LIN {X 0,Y 250.242,Z 442.898,A -85,B 0,C 180,E1 -18826.312,E2 -18826.312} C_VEL
LIN {X 0,Y 252.616,Z 436.287,A -85,B 0,C 180,E1 -18829.075,E2 -18829.075} C_VEL
LIN {X 0,Y 255.174,Z 429.183,A -85,B 0,C 180,E1 -18831.404,E2 -18831.404} C_VEL
LIN {X 0,Y 258.417,Z 420.356,A -85,B 0,C 180,E1 -18833.651,E2 -18833.651} C_VEL
LIN {X 0,Y 261.758,Z 410.378,A -85,B 0,C 180,E1 -18835.655,E2 -18835.655} C_VEL
LIN {X 0,Y 265.23,Z 399.079,A -85,B 0,C 180,E1 -18837.414,E2 -18837.414} C_VEL
LIN {X 0,Y 268.306,Z 387.871,A -85,B 0,C 180,E1 -18838.772,E2 -18838.772} C_VEL
LIN {X 0,Y 271.247,Z 375.163,A -85,B 0,C 180,E1 -18839.919,E2 -18839.919} C_VEL
LIN {X 0,Y 273.533,Z 362.414,A -85,B 0,C 180,E1 -18840.762,E2 -18840.762} C_VEL
LIN {X 0,Y 275.094,Z 349.012,A -85,B 0,C 180,E1 -18841.381,E2 -18841.381} C_VEL
LIN {X 0,Y 278.743,Z 306.37,A -85,B 0,C 180,E1 -18842.929,E2 -18842.929} C_VEL
LIN {X 0,Y 278.232,Z 292.635,A -85,B 0,C 180,E1 -18843.854,E2 -18843.854} C_VEL
LIN {X 0,Y 276.686,Z 276.192,A -85,B 0,C 180,E1 -18845.252,E2 -18845.252} C_VEL
LIN {X 0,Y 276.231,Z 273.561,A -85,B 0,C 180,E1 -18845.549,E2 -18845.549} C_VEL
LIN {X 0,Y 272.855,Z 266.156,A -85,B 0,C 180,E1 -18847.014,E2 -18847.014} C_VEL
LIN {X 0,Y 270.376,Z 261.218,A -85,B 0,C 180,E1 -18848.169,E2 -18848.169} C_VEL
LIN {X 0,Y 267.241,Z 255.568,A -85,B 0,C 180,E1 -18849.719,E2 -18849.719} C_VEL
LIN {X 0,Y 264.068,Z 250.117,A -85,B 0,C 180,E1 -18851.565,E2 -18851.565} C_VEL
LIN {X 0,Y 262.47,Z 244.735,A -85,B 0,C 180,E1 -18854.899,E2 -18854.899} C_VEL
LIN {X 0,Y 261.284,Z 241.259,A -85,B 0,C 180,E1 -18857.743,E2 -18857.743} C_VEL
LIN {X 0,Y 260.601,Z 239.385,A -85,B 0,C 180,E1 -18859.665,E2 -18859.665} C_VEL
LIN {X 0,Y 259.611,Z 236.801,A -85,B 0,C 180,E1 -18863.446,E2 -18863.446} C_VEL
LIN {X 0,Y 259.313,Z 236.04,A -85,B 0,C 180,E1 -18865.308,E2 -18865.308} C_VEL
LIN {X 0,Y 259.034,Z 235.596,A -85,B 0,C 180,E1 -18868.968,E2 -18868.968} C_VEL
LIN {X 0,Y 259.56,Z 236.51,A -85,B 0,C 180,E1 -18873.321,E2 -18873.321} C_VEL
LIN {X 0,Y 260.212,Z 238.641,A -85,B 0,C 180,E1 -18876.679,E2 -18876.679} C_VEL
LIN {X 0,Y 261.471,Z 242.04,A -85,B 0,C 180,E1 -18880.18,E2 -18880.18} C_VEL
LIN {X 0,Y 265.902,Z 248.153,A -85,B 0,C 180,E1 -18882.889,E2 -18882.889} C_VEL
LIN {X 0,Y 269.447,Z 253.421,A -85,B 0,C 180,E1 -18884.716,E2 -18884.716} C_VEL
LIN {X 0,Y 272.549,Z 258.468,A -85,B 0,C 180,E1 -18886.185,E2 -18886.185} C_VEL
LIN {X 0,Y 276.457,Z 265.391,A -85,B 0,C 180,E1 -18887.857,E2 -18887.857} C_VEL
LIN {X 0,Y 280.029,Z 273.175,A -85,B 0,C 180,E1 -18889.352,E2 -18889.352} C_VEL
LIN {X 0,Y 280.54,Z 277.359,A -85,B 0,C 180,E1 -18889.756,E2 -18889.756} C_VEL
LIN {X 0,Y 275.476,Z 327.139,A -85,B 0,C 180,E1 -18891.841,E2 -18891.841} C_VEL
LIN {X 0,Y 273.989,Z 339.798,A -85,B 0,C 180,E1 -18892.631,E2 -18892.631} C_VEL
LIN {X 0,Y 271.988,Z 352.049,A -85,B 0,C 180,E1 -18893.695,E2 -18893.695} C_VEL
LIN {X 0,Y 269.693,Z 362.869,A -85,B 0,C 180,E1 -18894.936,E2 -18894.936} C_VEL
LIN {X 0,Y 266.918,Z 373.483,A -85,B 0,C 180,E1 -18896.519,E2 -18896.519} C_VEL
LIN {X 0,Y 264.386,Z 381.823,A -85,B 0,C 180,E1 -18898.095,E2 -18898.095} C_VEL
LIN {X 0,Y 261.552,Z 389.85,A -85,B 0,C 180,E1 -18899.999,E2 -18899.999} C_VEL
LIN {X 0,Y 259.077,Z 396.31,A -85,B 0,C 180,E1 -18901.942,E2 -18901.942} C_VEL
LIN {X 0,Y 256.732,Z 401.481,A -85,B 0,C 180,E1 -18903.923,E2 -18903.923} C_VEL
LIN {X 0,Y 254.323,Z 406.197,A -85,B 0,C 180,E1 -18906.345,E2 -18906.345} C_VEL
LIN {X 0,Y 252.936,Z 408.542,A -85,B 0,C 180,E1 -18907.985,E2 -18907.985} C_VEL
LIN {X 0,Y 251.736,Z 410.331,A -85,B 0,C 180,E1 -18909.642,E2 -18909.642} C_VEL
LIN {X 0,Y 250.71,Z 411.505,A -85,B 0,C 180,E1 -18911.316,E2 -18911.316} C_VEL
LIN {X 0,Y 249.799,Z 412.162,A -85,B 0,C 180,E1 -18913.007,E2 -18913.007} C_VEL
LIN {X 0,Y 249.072,Z 412.229,A -85,B 0,C 180,E1 -18914.711,E2 -18914.711} C_VEL
LIN {X 0,Y 248.491,Z 411.75,A -85,B 0,C 180,E1 -18916.428,E2 -18916.428} C_VEL
LIN {X 0,Y 248.081,Z 410.706,A -85,B 0,C 180,E1 -18918.156,E2 -18918.156} C_VEL
LIN {X 0,Y 247.752,Z 408.241,A -85,B 0,C 180,E1 -18920.59,E2 -18920.59} C_VEL
LIN {X 0,Y 247.79,Z 403.869,A -85,B 0,C 180,E1 -18923.395,E2 -18923.395} C_VEL
LIN {X 0,Y 248.137,Z 398.052,A -85,B 0,C 180,E1 -18926.04,E2 -18926.04} C_VEL
LIN {X 0,Y 248.571,Z 391.701,A -85,B 0,C 180,E1 -18928.266,E2 -18928.266} C_VEL
LIN {X 0,Y 249.183,Z 383.577,A -85,B 0,C 180,E1 -18930.508,E2 -18930.508} C_VEL
LIN {X 0,Y 249.995,Z 374.485,A -85,B 0,C 180,E1 -18932.5,E2 -18932.5} C_VEL
LIN {X 0,Y 250.841,Z 364.034,A -85,B 0,C 180,E1 -18934.322,E2 -18934.322} C_VEL
LIN {X 0,Y 251.742,Z 352.485,A -85,B 0,C 180,E1 -18935.892,E2 -18935.892} C_VEL
LIN {X 0,Y 252.544,Z 339.639,A -85,B 0,C 180,E1 -18937.198,E2 -18937.198} C_VEL
LIN {X 0,Y 253.177,Z 325.928,A -85,B 0,C 180,E1 -18938.175,E2 -18938.175} C_VEL
LIN {X 0,Y 253.707,Z 305.907,A -85,B 0,C 180,E1 -18939.049,E2 -18939.049} C_VEL
LIN {X 0,Y 255.237,Z 260.217,A -85,B 0,C 180,E1 -18940.855,E2 -18940.855} C_VEL
LIN {X 0,Y 252.11,Z 234.672,A -85,B 0,C 180,E1 -18942.111,E2 -18942.111} C_VEL
LIN {X 0,Y 252.252,Z 229.715,A -85,B 0,C 180,E1 -18943.581,E2 -18943.581} C_VEL
LIN {X 0,Y 250.22,Z 219.034,A -85,B 0,C 180,E1 -18947.121,E2 -18947.121} C_VEL
LIN {X 0,Y 249.092,Z 213.695,A -85,B 0,C 180,E1 -18949.004,E2 -18949.004} C_VEL
LIN {X 0,Y 249.072,Z 213.461,A -85,B 0,C 180,E1 -18949.626,E2 -18949.626} C_VEL
LIN {X 0,Y 249.057,Z 213.463,A -85,B 0,C 180,E1 -18953.658,E2 -18953.658} C_VEL
LIN {X 0,Y 249.038,Z 213.464,A -85,B 0,C 180,E1 -18957.844,E2 -18957.844} C_VEL
LIN {X 0,Y 249.096,Z 213.458,A -85,B 0,C 180,E1 -18961.337,E2 -18961.337} C_VEL
LIN {X 0,Y 249.151,Z 213.448,A -85,B 0,C 180,E1 -18964.967,E2 -18964.967} C_VEL
LIN {X 0,Y 249.109,Z 213.453,A -85,B 0,C 180,E1 -18970.21,E2 -18970.21} C_VEL
LIN {X 0,Y 249.241,Z 213.437,A -85,B 0,C 180,E1 -18973.621,E2 -18973.621} C_VEL
LIN {X 0,Y 249.251,Z 213.435,A -85,B 0,C 180,E1 -18978.615,E2 -18978.615} C_VEL
LIN {X 0,Y 249.482,Z 213.405,A -85,B 0,C 180,E1 -18981.902,E2 -18981.902} C_VEL
LIN {X 0,Y 249.435,Z 213.414,A -85,B 0,C 180,E1 -18986.768,E2 -18986.768} C_VEL
LIN {X 0,Y 249.726,Z 213.374,A -85,B 0,C 180,E1 -18989.999,E2 -18989.999} C_VEL
LIN {X 0,Y 249.434,Z 213.415,A -85,B 0,C 180,E1 -18993.229,E2 -18993.229} C_VEL
LIN {X 0,Y 249.476,Z 213.404,A -85,B 0,C 180,E1 -18998.096,E2 -18998.096} C_VEL
LIN {X 0,Y 249.249,Z 213.436,A -85,B 0,C 180,E1 -19001.382,E2 -19001.382} C_VEL
LIN {X 0,Y 249.238,Z 213.436,A -85,B 0,C 180,E1 -19006.377,E2 -19006.377} C_VEL
LIN {X 0,Y 249.082,Z 213.456,A -85,B 0,C 180,E1 -19011.517,E2 -19011.517} C_VEL
LIN {X 0,Y 249.126,Z 213.449,A -85,B 0,C 180,E1 -19015.482,E2 -19015.482} C_VEL
LIN {X 0,Y 249.078,Z 213.458,A -85,B 0,C 180,E1 -19018.993,E2 -19018.993} C_VEL
LIN {X 0,Y 249.03,Z 213.465,A -85,B 0,C 180,E1 -19022.424,E2 -19022.424} C_VEL
LIN {X 0,Y 249.069,Z 213.46,A -85,B 0,C 180,E1 -19026.337,E2 -19026.337} C_VEL
LIN {X 0,Y 249.071,Z 213.459,A -85,B 0,C 180,E1 -19030.463,E2 -19030.463} C_VEL
LIN {X 0,Y 249.015,Z 213.465,A -85,B 0,C 180,E1 -19034.874,E2 -19034.874} C_VEL
LIN {X 0,Y 249.047,Z 213.46,A -85,B 0,C 180,E1 -19037.37,E2 -19037.37} C_VEL
LIN {X 0,Y 249.058,Z 213.462,A -85,B 0,C 180,E1 -19042.193,E2 -19042.193} C_VEL
LIN {X 0,Y 249.055,Z 213.46,A -85,B 0,C 180,E1 -19045.642,E2 -19045.642} C_VEL
LIN {X 0,Y 249.044,Z 213.459,A -85,B 0,C 180,E1 -19049.473,E2 -19049.473} C_VEL
LIN {X 0,Y 249.066,Z 213.458,A -85,B 0,C 180,E1 -19053.162,E2 -19053.162} C_VEL
LIN {X 0,Y 249.072,Z 213.455,A -85,B 0,C 180,E1 -19056.733,E2 -19056.733} C_VEL
LIN {X 0,Y 249.104,Z 213.456,A -85,B 0,C 180,E1 -19060.212,E2 -19060.212} C_VEL
LIN {X 0,Y 249.235,Z 213.439,A -85,B 0,C 180,E1 -19063.622,E2 -19063.622} C_VEL
LIN {X 0,Y 249.237,Z 213.437,A -85,B 0,C 180,E1 -19068.617,E2 -19068.617} C_VEL
LIN {X 0,Y 249.448,Z 213.413,A -85,B 0,C 180,E1 -19071.903,E2 -19071.903} C_VEL
LIN {X 0,Y 249.289,Z 213.429,A -85,B 0,C 180,E1 -19075.149,E2 -19075.149} C_VEL
LIN {X 0,Y 249.669,Z 213.383,A -85,B 0,C 180,E1 -19078.388,E2 -19078.388} C_VEL
LIN {X 0,Y 249.669,Z 213.385,A -85,B 0,C 180,E1 -19081.614,E2 -19081.614} C_VEL
LIN {X 0,Y 249.454,Z 213.41,A -85,B 0,C 180,E1 -19086.471,E2 -19086.471} C_VEL
LIN {X 0,Y 249.383,Z 213.419,A -85,B 0,C 180,E1 -19089.736,E2 -19089.736} C_VEL
LIN {X 0,Y 249.2,Z 213.442,A -85,B 0,C 180,E1 -19094.704,E2 -19094.704} C_VEL
LIN {X 0,Y 249.134,Z 213.448,A -85,B 0,C 180,E1 -19098.078,E2 -19098.078} C_VEL
LIN {X 0,Y 249.082,Z 213.459,A -85,B 0,C 180,E1 -19101.519,E2 -19101.519} C_VEL
LIN {X 0,Y 249.073,Z 213.457,A -85,B 0,C 180,E1 -19103.868,E2 -19103.868} C_VEL
LIN {X 0,Y 248.416,Z 213.543,A -85,B 0,C 180,E1 -19105.217,E2 -19105.217} C_VEL
LIN {X 0,Y 245.523,Z 213.901,A -85,B 0,C 180,E1 -19107.414,E2 -19107.414} C_VEL
LIN {X 0,Y 243.064,Z 214.209,A -85,B 0,C 180,E1 -19109.205,E2 -19109.205} C_VEL
LIN {X 0,Y 242.026,Z 214.336,A -85,B 0,C 180,E1 -19110.595,E2 -19110.595} C_VEL
LIN {X 0,Y 241.952,Z 214.342,A -85,B 0,C 180,E1 -19111.066,E2 -19111.066} C_VEL
LIN {X 0,Y 242.002,Z 214.339,A -85,B 0,C 180,E1 -19115.598,E2 -19115.598} C_VEL
LIN {X 0,Y 241.953,Z 214.345,A -85,B 0,C 180,E1 -19119.721,E2 -19119.721} C_VEL
LIN {X 0,Y 241.916,Z 214.349,A -85,B 0,C 180,E1 -19124.206,E2 -19124.206} C_VEL
LIN {X 0,Y 241.932,Z 214.348,A -85,B 0,C 180,E1 -19128.079,E2 -19128.079} C_VEL
LIN {X 0,Y 242.039,Z 214.525,A -85,B 0,C 180,E1 -19132.235,E2 -19132.235} C_VEL
LIN {X 0,Y 245.004,Z 227.718,A -85,B 0,C 180,E1 -19136.293,E2 -19136.293} C_VEL
LIN {X 0,Y 247.94,Z 241.383,A -85,B 0,C 180,E1 -19140.263,E2 -19140.263} C_VEL
LIN {X 0,Y 248.195,Z 243.179,A -85,B 0,C 180,E1 -19140.762,E2 -19140.762} C_VEL
LIN {X 0,Y 246.035,Z 256.439,A -85,B 0,C 180,E1 -19144.177,E2 -19144.177} C_VEL
LIN {X 0,Y 247.085,Z 277.97,A -85,B 0,C 180,E1 -19145.106,E2 -19145.106} C_VEL
LIN {X 0,Y 248.735,Z 300.915,A -85,B 0,C 180,E1 -19146.066,E2 -19146.066} C_VEL
LIN {X 0,Y 247.023,Z 359.054,A -85,B 0,C 180,E1 -19148.24,E2 -19148.24} C_VEL
LIN {X 0,Y 246.323,Z 371.481,A -85,B 0,C 180,E1 -19148.998,E2 -19148.998} C_VEL
LIN {X 0,Y 245.403,Z 383.203,A -85,B 0,C 180,E1 -19150.01,E2 -19150.01} C_VEL
LIN {X 0,Y 244.335,Z 394.661,A -85,B 0,C 180,E1 -19151.339,E2 -19151.339} C_VEL
LIN {X 0,Y 243.271,Z 405.628,A -85,B 0,C 180,E1 -19152.962,E2 -19152.962} C_VEL
LIN {X 0,Y 242.195,Z 415.752,A -85,B 0,C 180,E1 -19154.862,E2 -19154.862} C_VEL
LIN {X 0,Y 241.442,Z 424.766,A -85,B 0,C 180,E1 -19156.964,E2 -19156.964} C_VEL
LIN {X 0,Y 240.968,Z 432.123,A -85,B 0,C 180,E1 -19159.073,E2 -19159.073} C_VEL
LIN {X 0,Y 240.761,Z 439.176,A -85,B 0,C 180,E1 -19161.609,E2 -19161.609} C_VEL
LIN {X 0,Y 240.805,Z 444.675,A -85,B 0,C 180,E1 -19164.138,E2 -19164.138} C_VEL
LIN {X 0,Y 240.983,Z 448.811,A -85,B 0,C 180,E1 -19166.657,E2 -19166.657} C_VEL
LIN {X 0,Y 241.109,Z 450.863,A -85,B 0,C 180,E1 -19168.331,E2 -19168.331} C_VEL
LIN {X 0,Y 241.116,Z 452.378,A -85,B 0,C 180,E1 -19170.001,E2 -19170.001} C_VEL
LIN {X 0,Y 240.997,Z 453.423,A -85,B 0,C 180,E1 -19171.672,E2 -19171.672} C_VEL
LIN {X 0,Y 240.622,Z 453.947,A -85,B 0,C 180,E1 -19173.35,E2 -19173.35} C_VEL
LIN {X 0,Y 240.281,Z 453.905,A -85,B 0,C 180,E1 -19176.022,E2 -19176.022} C_VEL
LIN {X 0,Y 240.213,Z 452.989,A -85,B 0,C 180,E1 -19178.413,E2 -19178.413} C_VEL
LIN {X 0,Y 240.738,Z 450.239,A -85,B 0,C 180,E1 -19181.793,E2 -19181.793} C_VEL
LIN {X 0,Y 241.879,Z 447.064,A -85,B 0,C 180,E1 -19184.3,E2 -19184.3} C_VEL
LIN {X 0,Y 243.423,Z 442.874,A -85,B 0,C 180,E1 -19186.782,E2 -19186.782} C_VEL
LIN {X 0,Y 245.831,Z 436.744,A -85,B 0,C 180,E1 -19189.547,E2 -19189.547} C_VEL
LIN {X 0,Y 248.587,Z 429.654,A -85,B 0,C 180,E1 -19192.001,E2 -19192.001} C_VEL
LIN {X 0,Y 251.986,Z 421.175,A -85,B 0,C 180,E1 -19194.293,E2 -19194.293} C_VEL
LIN {X 0,Y 255.123,Z 412.586,A -85,B 0,C 180,E1 -19196.153,E2 -19196.153} C_VEL
LIN {X 0,Y 258.683,Z 402.079,A -85,B 0,C 180,E1 -19197.948,E2 -19197.948} C_VEL
LIN {X 0,Y 261.804,Z 391.752,A -85,B 0,C 180,E1 -19199.336,E2 -19199.336} C_VEL
LIN {X 0,Y 265.258,Z 378.523,A -85,B 0,C 180,E1 -19200.667,E2 -19200.667} C_VEL
LIN {X 0,Y 267.695,Z 366.659,A -85,B 0,C 180,E1 -19201.564,E2 -19201.564} C_VEL
LIN {X 0,Y 269.831,Z 352.408,A -85,B 0,C 180,E1 -19202.328,E2 -19202.328} C_VEL
LIN {X 0,Y 273.994,Z 306.663,A -85,B 0,C 180,E1 -19204.05,E2 -19204.05} C_VEL
LIN {X 0,Y 273.515,Z 292.928,A -85,B 0,C 180,E1 -19205.03,E2 -19205.03} C_VEL
LIN {X 0,Y 272.25,Z 277.749,A -85,B 0,C 180,E1 -19206.404,E2 -19206.404} C_VEL
LIN {X 0,Y 269.163,Z 270.902,A -85,B 0,C 180,E1 -19207.837,E2 -19207.837} C_VEL
LIN {X 0,Y 266.967,Z 266.304,A -85,B 0,C 180,E1 -19208.942,E2 -19208.942} C_VEL
LIN {X 0,Y 264.32,Z 261.353,A -85,B 0,C 180,E1 -19210.347,E2 -19210.347} C_VEL
LIN {X 0,Y 260.674,Z 255.2,A -85,B 0,C 180,E1 -19212.513,E2 -19212.513} C_VEL
LIN {X 0,Y 256.954,Z 248.907,A -85,B 0,C 180,E1 -19215.328,E2 -19215.328} C_VEL
LIN {X 0,Y 255.623,Z 245.043,A -85,B 0,C 180,E1 -19218.711,E2 -19218.711} C_VEL
LIN {X 0,Y 254.553,Z 242.132,A -85,B 0,C 180,E1 -19222.597,E2 -19222.597} C_VEL
LIN {X 0,Y 254.253,Z 241.129,A -85,B 0,C 180,E1 -19224.515,E2 -19224.515} C_VEL
LIN {X 0,Y 253.852,Z 240.45,A -85,B 0,C 180,E1 -19229.122,E2 -19229.122} C_VEL
LIN {X 0,Y 254.111,Z 240.979,A -85,B 0,C 180,E1 -19232.256,E2 -19232.256} C_VEL
LIN {X 0,Y 254.384,Z 241.552,A -85,B 0,C 180,E1 -19233.765,E2 -19233.765} C_VEL
LIN {X 0,Y 255.017,Z 243.339,A -85,B 0,C 180,E1 -19236.387,E2 -19236.387} C_VEL
LIN {X 0,Y 259.406,Z 248.969,A -85,B 0,C 180,E1 -19239.974,E2 -19239.974} C_VEL
LIN {X 0,Y 263.342,Z 254.427,A -85,B 0,C 180,E1 -19242.435,E2 -19242.435} C_VEL
LIN {X 0,Y 266.413,Z 259.247,A -85,B 0,C 180,E1 -19244.128,E2 -19244.128} C_VEL
LIN {X 0,Y 269.216,Z 263.882,A -85,B 0,C 180,E1 -19245.514,E2 -19245.514} C_VEL
LIN {X 0,Y 273.059,Z 271.072,A -85,B 0,C 180,E1 -19247.297,E2 -19247.297} C_VEL
LIN {X 0,Y 275.758,Z 277.511,A -85,B 0,C 180,E1 -19248.545,E2 -19248.545} C_VEL
LIN {X 0,Y 275.789,Z 279.841,A -85,B 0,C 180,E1 -19248.723,E2 -19248.723} C_VEL
LIN {X 0,Y 270.622,Z 328.589,A -85,B 0,C 180,E1 -19250.802,E2 -19250.802} C_VEL
LIN {X 0,Y 268.929,Z 341.564,A -85,B 0,C 180,E1 -19251.641,E2 -19251.641} C_VEL
LIN {X 0,Y 266.965,Z 352.562,A -85,B 0,C 180,E1 -19252.626,E2 -19252.626} C_VEL
LIN {X 0,Y 264.468,Z 363.457,A -85,B 0,C 180,E1 -19253.897,E2 -19253.897} C_VEL
LIN {X 0,Y 261.219,Z 375.14,A -85,B 0,C 180,E1 -19255.676,E2 -19255.676} C_VEL
LIN {X 0,Y 258.565,Z 383.268,A -85,B 0,C 180,E1 -19257.273,E2 -19257.273} C_VEL
LIN {X 0,Y 255.535,Z 391.182,A -85,B 0,C 180,E1 -19259.211,E2 -19259.211} C_VEL
LIN {X 0,Y 253.054,Z 397.105,A -85,B 0,C 180,E1 -19261.065,E2 -19261.065} C_VEL
LIN {X 0,Y 250.411,Z 402.538,A -85,B 0,C 180,E1 -19263.217,E2 -19263.217} C_VEL
LIN {X 0,Y 248.03,Z 406.89,A -85,B 0,C 180,E1 -19265.509,E2 -19265.509} C_VEL
LIN {X 0,Y 245.68,Z 410.416,A -85,B 0,C 180,E1 -19268.222,E2 -19268.222} C_VEL
LIN {X 0,Y 244.462,Z 411.843,A -85,B 0,C 180,E1 -19269.932,E2 -19269.932} C_VEL
LIN {X 0,Y 243.43,Z 412.692,A -85,B 0,C 180,E1 -19271.659,E2 -19271.659} C_VEL
LIN {X 0,Y 242.549,Z 413.034,A -85,B 0,C 180,E1 -19273.402,E2 -19273.402} C_VEL
LIN {X 0,Y 241.491,Z 412.383,A -85,B 0,C 180,E1 -19276.18,E2 -19276.18} C_VEL
LIN {X 0,Y 240.877,Z 410.594,A -85,B 0,C 180,E1 -19278.719,E2 -19278.719} C_VEL
LIN {X 0,Y 240.632,Z 407.265,A -85,B 0,C 180,E1 -19281.493,E2 -19281.493} C_VEL
LIN {X 0,Y 240.773,Z 402.698,A -85,B 0,C 180,E1 -19284.119,E2 -19284.119} C_VEL
LIN {X 0,Y 241.108,Z 397.438,A -85,B 0,C 180,E1 -19286.392,E2 -19286.392} C_VEL
LIN {X 0,Y 241.669,Z 389.71,A -85,B 0,C 180,E1 -19288.984,E2 -19288.984} C_VEL
LIN {X 0,Y 242.241,Z 382.109,A -85,B 0,C 180,E1 -19290.995,E2 -19290.995} C_VEL
LIN {X 0,Y 243.1,Z 372.57,A -85,B 0,C 180,E1 -19293.029,E2 -19293.029} C_VEL
LIN {X 0,Y 244.04,Z 361.305,A -85,B 0,C 180,E1 -19294.915,E2 -19294.915} C_VEL
LIN {X 0,Y 244.911,Z 349.633,A -85,B 0,C 180,E1 -19296.422,E2 -19296.422} C_VEL
LIN {X 0,Y 245.629,Z 337.82,A -85,B 0,C 180,E1 -19297.574,E2 -19297.574} C_VEL
LIN {X 0,Y 246.218,Z 324.894,A -85,B 0,C 180,E1 -19298.473,E2 -19298.473} C_VEL
LIN {X 0,Y 246.945,Z 299.704,A -85,B 0,C 180,E1 -19299.574,E2 -19299.574} C_VEL
LIN {X 0,Y 248.312,Z 260.898,A -85,B 0,C 180,E1 -19301.163,E2 -19301.163} C_VEL
LIN {X 0,Y 245.18,Z 235.277,A -85,B 0,C 180,E1 -19302.436,E2 -19302.436} C_VEL
LIN {X 0,Y 245.269,Z 233.089,A -85,B 0,C 180,E1 -19302.999,E2 -19302.999} C_VEL
LIN {X 0,Y 245.025,Z 229.434,A -85,B 0,C 180,E1 -19304.186,E2 -19304.186} C_VEL
LIN {X 0,Y 242.968,Z 219.033,A -85,B 0,C 180,E1 -19307.737,E2 -19307.737} C_VEL
LIN {X 0,Y 242.072,Z 214.513,A -85,B 0,C 180,E1 -19309.394,E2 -19309.394} C_VEL
LIN {X 0,Y 241.99,Z 214.341,A -85,B 0,C 180,E1 -19312.417,E2 -19312.417} C_VEL
LIN {X 0,Y 241.987,Z 214.341,A -85,B 0,C 180,E1 -19316.507,E2 -19316.507} C_VEL
LIN {X 0,Y 242.036,Z 214.334,A -85,B 0,C 180,E1 -19320.586,E2 -19320.586} C_VEL
LIN {X 0,Y 242.067,Z 214.33,A -85,B 0,C 180,E1 -19324.182,E2 -19324.182} C_VEL
LIN {X 0,Y 242.052,Z 214.331,A -85,B 0,C 180,E1 -19328.296,E2 -19328.296} C_VEL
LIN {X 0,Y 242.162,Z 214.32,A -85,B 0,C 180,E1 -19333.277,E2 -19333.277} C_VEL
LIN {X 0,Y 242.185,Z 214.315,A -85,B 0,C 180,E1 -19338.279,E2 -19338.279} C_VEL
LIN {X 0,Y 242.433,Z 214.284,A -85,B 0,C 180,E1 -19341.665,E2 -19341.665} C_VEL
LIN {X 0,Y 242.26,Z 214.309,A -85,B 0,C 180,E1 -19345.006,E2 -19345.006} C_VEL
LIN {X 0,Y 242.634,Z 214.258,A -85,B 0,C 180,E1 -19348.339,E2 -19348.339} C_VEL
LIN {X 0,Y 242.634,Z 214.259,A -85,B 0,C 180,E1 -19351.659,E2 -19351.659} C_VEL
LIN {X 0,Y 242.428,Z 214.286,A -85,B 0,C 180,E1 -19356.658,E2 -19356.658} C_VEL
LIN {X 0,Y 242.311,Z 214.299,A -85,B 0,C 180,E1 -19360.021,E2 -19360.021} C_VEL
LIN {X 0,Y 242.163,Z 214.318,A -85,B 0,C 180,E1 -19365.14,E2 -19365.14} C_VEL
LIN {X 0,Y 242.069,Z 214.331,A -85,B 0,C 180,E1 -19368.623,E2 -19368.623} C_VEL
LIN {X 0,Y 242.008,Z 214.338,A -85,B 0,C 180,E1 -19372.179,E2 -19372.179} C_VEL
LIN {X 0,Y 242.061,Z 214.329,A -85,B 0,C 180,E1 -19375.837,E2 -19375.837} C_VEL
LIN {X 0,Y 242.025,Z 214.335,A -85,B 0,C 180,E1 -19379.579,E2 -19379.579} C_VEL
LIN {X 0,Y 241.985,Z 214.338,A -85,B 0,C 180,E1 -19383.49,E2 -19383.49} C_VEL
LIN {X 0,Y 242.007,Z 214.337,A -85,B 0,C 180,E1 -19387.577,E2 -19387.577} C_VEL
LIN {X 0,Y 241.978,Z 214.339,A -85,B 0,C 180,E1 -19391.912,E2 -19391.912} C_VEL
LIN {X 0,Y 241.98,Z 214.343,A -85,B 0,C 180,E1 -19396.558,E2 -19396.558} C_VEL
LIN {X 0,Y 241.975,Z 214.343,A -85,B 0,C 180,E1 -19400.286,E2 -19400.286} C_VEL
LIN {X 0,Y 242.03,Z 214.337,A -85,B 0,C 180,E1 -19404.497,E2 -19404.497} C_VEL
LIN {X 0,Y 241.969,Z 214.342,A -85,B 0,C 180,E1 -19408.48,E2 -19408.48} C_VEL
LIN {X 0,Y 242,Z 214.341,A -85,B 0,C 180,E1 -19412.313,E2 -19412.313} C_VEL
LIN {X 0,Y 242.05,Z 214.334,A -85,B 0,C 180,E1 -19416.016,E2 -19416.016} C_VEL
LIN {X 0,Y 242.03,Z 214.335,A -85,B 0,C 180,E1 -19419.608,E2 -19419.608} C_VEL
LIN {X 0,Y 242.156,Z 214.319,A -85,B 0,C 180,E1 -19423.279,E2 -19423.279} C_VEL
LIN {X 0,Y 242.174,Z 214.318,A -85,B 0,C 180,E1 -19428.28,E2 -19428.28} C_VEL
LIN {X 0,Y 242.393,Z 214.292,A -85,B 0,C 180,E1 -19431.665,E2 -19431.665} C_VEL
LIN {X 0,Y 242.25,Z 214.306,A -85,B 0,C 180,E1 -19435.008,E2 -19435.008} C_VEL
LIN {X 0,Y 242.629,Z 214.26,A -85,B 0,C 180,E1 -19438.341,E2 -19438.341} C_VEL
LIN {X 0,Y 242.629,Z 214.261,A -85,B 0,C 180,E1 -19441.661,E2 -19441.661} C_VEL
LIN {X 0,Y 242.427,Z 214.285,A -85,B 0,C 180,E1 -19446.66,E2 -19446.66} C_VEL
LIN {X 0,Y 242.308,Z 214.298,A -85,B 0,C 180,E1 -19450.023,E2 -19450.023} C_VEL
LIN {X 0,Y 242.161,Z 214.32,A -85,B 0,C 180,E1 -19455.142,E2 -19455.142} C_VEL
LIN {X 0,Y 242.068,Z 214.328,A -85,B 0,C 180,E1 -19458.625,E2 -19458.625} C_VEL
LIN {X 0,Y 242.008,Z 214.337,A -85,B 0,C 180,E1 -19462.181,E2 -19462.181} C_VEL
LIN {X 0,Y 242.062,Z 214.33,A -85,B 0,C 180,E1 -19465.839,E2 -19465.839} C_VEL
LIN {X 0,Y 242.003,Z 214.34,A -85,B 0,C 180,E1 -19469.585,E2 -19469.585} C_VEL
LIN {X 0,Y 241.952,Z 214.342,A -85,B 0,C 180,E1 -19471.066,E2 -19471.066} C_VEL
LIN {X 0,Y 241.297,Z 214.428,A -85,B 0,C 180,E1 -19472.456,E2 -19472.456} C_VEL
LIN {X 0,Y 238.411,Z 214.787,A -85,B 0,C 180,E1 -19474.722,E2 -19474.722} C_VEL
LIN {X 0,Y 235.968,Z 215.09,A -85,B 0,C 180,E1 -19476.569,E2 -19476.569} C_VEL
LIN {X 0,Y 234.953,Z 215.216,A -85,B 0,C 180,E1 -19478.003,E2 -19478.003} C_VEL
LIN {X 0,Y 234.89,Z 215.223,A -85,B 0,C 180,E1 -19478.489,E2 -19478.489} C_VEL
LIN {X 0,Y 234.878,Z 215.227,A -85,B 0,C 180,E1 -19481.581,E2 -19481.581} C_VEL
LIN {X 0,Y 234.882,Z 215.226,A -85,B 0,C 180,E1 -19485.9,E2 -19485.9} C_VEL
LIN {X 0,Y 234.88,Z 215.229,A -85,B 0,C 180,E1 -19488.834,E2 -19488.834} C_VEL
LIN {X 0,Y 234.993,Z 215.432,A -85,B 0,C 180,E1 -19491.819,E2 -19491.819} C_VEL
LIN {X 0,Y 237.844,Z 228.125,A -85,B 0,C 180,E1 -19495.847,E2 -19495.847} C_VEL
LIN {X 0,Y 240.65,Z 241.145,A -85,B 0,C 180,E1 -19499.752,E2 -19499.752} C_VEL
LIN {X 0,Y 241.062,Z 244.801,A -85,B 0,C 180,E1 -19500.796,E2 -19500.796} C_VEL
LIN {X 0,Y 239.126,Z 256.051,A -85,B 0,C 180,E1 -19503.785,E2 -19503.785} C_VEL
LIN {X 0,Y 240.01,Z 276.708,A -85,B 0,C 180,E1 -19504.714,E2 -19504.714} C_VEL
LIN {X 0,Y 241.754,Z 301.362,A -85,B 0,C 180,E1 -19505.791,E2 -19505.791} C_VEL
LIN {X 0,Y 239.987,Z 358.705,A -85,B 0,C 180,E1 -19508.021,E2 -19508.021} C_VEL
LIN {X 0,Y 239.29,Z 371.062,A -85,B 0,C 180,E1 -19508.802,E2 -19508.802} C_VEL
LIN {X 0,Y 238.473,Z 381.707,A -85,B 0,C 180,E1 -19509.741,E2 -19509.741} C_VEL
LIN {X 0,Y 237.324,Z 393.659,A -85,B 0,C 180,E1 -19511.142,E2 -19511.142} C_VEL
LIN {X 0,Y 236.195,Z 405.3,A -85,B 0,C 180,E1 -19512.914,E2 -19512.914} C_VEL
LIN {X 0,Y 235.134,Z 415.219,A -85,B 0,C 180,E1 -19514.84,E2 -19514.84} C_VEL
LIN {X 0,Y 234.387,Z 424.22,A -85,B 0,C 180,E1 -19517.005,E2 -19517.005} C_VEL
LIN {X 0,Y 233.925,Z 431.56,A -85,B 0,C 180,E1 -19519.178,E2 -19519.178} C_VEL
LIN {X 0,Y 233.723,Z 438.587,A -85,B 0,C 180,E1 -19521.79,E2 -19521.79} C_VEL
LIN {X 0,Y 233.769,Z 443.252,A -85,B 0,C 180,E1 -19523.961,E2 -19523.961} C_VEL
LIN {X 0,Y 233.966,Z 447.567,A -85,B 0,C 180,E1 -19526.557,E2 -19526.557} C_VEL
LIN {X 0,Y 234.069,Z 449.75,A -85,B 0,C 180,E1 -19528.281,E2 -19528.281} C_VEL
LIN {X 0,Y 234.083,Z 451.357,A -85,B 0,C 180,E1 -19530.001,E2 -19530.001} C_VEL
LIN {X 0,Y 233.944,Z 452.461,A -85,B 0,C 180,E1 -19531.723,E2 -19531.723} C_VEL
LIN {X 0,Y 233.568,Z 453.099,A -85,B 0,C 180,E1 -19533.451,E2 -19533.451} C_VEL
LIN {X 0,Y 233.224,Z 453.225,A -85,B 0,C 180,E1 -19536.045,E2 -19536.045} C_VEL
LIN {X 0,Y 233.157,Z 452.402,A -85,B 0,C 180,E1 -19538.669,E2 -19538.669} C_VEL
LIN {X 0,Y 233.36,Z 451.359,A -85,B 0,C 180,E1 -19540.412,E2 -19540.412} C_VEL
LIN {X 0,Y 233.742,Z 449.87,A -85,B 0,C 180,E1 -19542.151,E2 -19542.151} C_VEL
LIN {X 0,Y 234.965,Z 446.886,A -85,B 0,C 180,E1 -19544.73,E2 -19544.73} C_VEL
LIN {X 0,Y 236.627,Z 442.873,A -85,B 0,C 180,E1 -19547.279,E2 -19547.279} C_VEL
LIN {X 0,Y 238.829,Z 437.678,A -85,B 0,C 180,E1 -19549.806,E2 -19549.806} C_VEL
LIN {X 0,Y 242.037,Z 430.2,A -85,B 0,C 180,E1 -19552.628,E2 -19552.628} C_VEL
LIN {X 0,Y 245.589,Z 422.035,A -85,B 0,C 180,E1 -19554.968,E2 -19554.968} C_VEL
LIN {X 0,Y 248.87,Z 413.774,A -85,B 0,C 180,E1 -19556.862,E2 -19556.862} C_VEL
LIN {X 0,Y 252.527,Z 403.736,A -85,B 0,C 180,E1 -19558.692,E2 -19558.692} C_VEL
LIN {X 0,Y 256.173,Z 392.632,A -85,B 0,C 180,E1 -19560.273,E2 -19560.273} C_VEL
LIN {X 0,Y 259.339,Z 381.873,A -85,B 0,C 180,E1 -19561.445,E2 -19561.445} C_VEL
LIN {X 0,Y 262.309,Z 368.985,A -85,B 0,C 180,E1 -19562.517,E2 -19562.517} C_VEL
LIN {X 0,Y 264.556,Z 356.138,A -85,B 0,C 180,E1 -19563.281,E2 -19563.281} C_VEL
LIN {X 0,Y 266.971,Z 333.427,A -85,B 0,C 180,E1 -19564.175,E2 -19564.175} C_VEL
LIN {X 0,Y 269.438,Z 307.883,A -85,B 0,C 180,E1 -19565.167,E2 -19565.167} C_VEL
LIN {X 0,Y 269.118,Z 294.607,A -85,B 0,C 180,E1 -19566.158,E2 -19566.158} C_VEL
LIN {X 0,Y 268.15,Z 281.712,A -85,B 0,C 180,E1 -19567.354,E2 -19567.354} C_VEL
LIN {X 0,Y 264.649,Z 273.323,A -85,B 0,C 180,E1 -19569.208,E2 -19569.208} C_VEL
LIN {X 0,Y 261.35,Z 266.949,A -85,B 0,C 180,E1 -19571.058,E2 -19571.058} C_VEL
LIN {X 0,Y 258.273,Z 261.5,A -85,B 0,C 180,E1 -19573.003,E2 -19573.003} C_VEL
LIN {X 0,Y 254.352,Z 254.93,A -85,B 0,C 180,E1 -19576.038,E2 -19576.038} C_VEL
LIN {X 0,Y 251.07,Z 250.024,A -85,B 0,C 180,E1 -19579.549,E2 -19579.549} C_VEL
LIN {X 0,Y 249.498,Z 247.198,A -85,B 0,C 180,E1 -19582.434,E2 -19582.434} C_VEL
LIN {X 0,Y 249.03,Z 245.889,A -85,B 0,C 180,E1 -19584.928,E2 -19584.928} C_VEL
LIN {X 0,Y 248.775,Z 245.426,A -85,B 0,C 180,E1 -19588.718,E2 -19588.718} C_VEL
LIN {X 0,Y 249.865,Z 246.591,A -85,B 0,C 180,E1 -19591.909,E2 -19591.909} C_VEL
LIN {X 0,Y 252.858,Z 249.7,A -85,B 0,C 180,E1 -19595.812,E2 -19595.812} C_VEL
LIN {X 0,Y 257.209,Z 255.47,A -85,B 0,C 180,E1 -19599.574,E2 -19599.574} C_VEL
LIN {X 0,Y 260.693,Z 260.568,A -85,B 0,C 180,E1 -19601.898,E2 -19601.898} C_VEL
LIN {X 0,Y 263.913,Z 265.887,A -85,B 0,C 180,E1 -19603.792,E2 -19603.792} C_VEL
LIN {X 0,Y 266.213,Z 269.891,A -85,B 0,C 180,E1 -19604.986,E2 -19604.986} C_VEL
LIN {X 0,Y 269.463,Z 276.342,A -85,B 0,C 180,E1 -19606.627,E2 -19606.627} C_VEL
LIN {X 0,Y 271.419,Z 280.946,A -85,B 0,C 180,E1 -19607.564,E2 -19607.564} C_VEL
LIN {X 0,Y 265.924,Z 329.453,A -85,B 0,C 180,E1 -19609.682,E2 -19609.682} C_VEL
LIN {X 0,Y 264.207,Z 341.756,A -85,B 0,C 180,E1 -19610.488,E2 -19610.488} C_VEL
LIN {X 0,Y 262.221,Z 352.548,A -85,B 0,C 180,E1 -19611.445,E2 -19611.445} C_VEL
LIN {X 0,Y 259.444,Z 364.16,A -85,B 0,C 180,E1 -19612.802,E2 -19612.802} C_VEL
LIN {X 0,Y 256.534,Z 374.047,A -85,B 0,C 180,E1 -19614.3,E2 -19614.3} C_VEL
LIN {X 0,Y 253.438,Z 383.063,A -85,B 0,C 180,E1 -19616.034,E2 -19616.034} C_VEL
LIN {X 0,Y 250.194,Z 391.101,A -85,B 0,C 180,E1 -19617.987,E2 -19617.987} C_VEL
LIN {X 0,Y 247.326,Z 397.584,A -85,B 0,C 180,E1 -19619.999,E2 -19619.999} C_VEL
LIN {X 0,Y 244.152,Z 403.662,A -85,B 0,C 180,E1 -19622.474,E2 -19622.474} C_VEL
LIN {X 0,Y 241.385,Z 408.2,A -85,B 0,C 180,E1 -19625.01,E2 -19625.01} C_VEL
LIN {X 0,Y 239.776,Z 410.434,A -85,B 0,C 180,E1 -19626.732,E2 -19626.732} C_VEL
LIN {X 0,Y 238.395,Z 412.097,A -85,B 0,C 180,E1 -19628.476,E2 -19628.476} C_VEL
LIN {X 0,Y 236.524,Z 413.573,A -85,B 0,C 180,E1 -19631.315,E2 -19631.315} C_VEL
LIN {X 0,Y 235.279,Z 413.719,A -85,B 0,C 180,E1 -19633.825,E2 -19633.825} C_VEL
LIN {X 0,Y 234.346,Z 412.806,A -85,B 0,C 180,E1 -19636.325,E2 -19636.325} C_VEL
LIN {X 0,Y 233.701,Z 410.287,A -85,B 0,C 180,E1 -19639.316,E2 -19639.316} C_VEL
LIN {X 0,Y 233.53,Z 406.541,A -85,B 0,C 180,E1 -19642.097,E2 -19642.097} C_VEL
LIN {X 0,Y 233.756,Z 401.223,A -85,B 0,C 180,E1 -19644.892,E2 -19644.892} C_VEL
LIN {X 0,Y 234.141,Z 395.375,A -85,B 0,C 180,E1 -19647.241,E2 -19647.241} C_VEL
LIN {X 0,Y 234.747,Z 387.462,A -85,B 0,C 180,E1 -19649.746,E2 -19649.746} C_VEL
LIN {X 0,Y 235.517,Z 378.43,A -85,B 0,C 180,E1 -19651.982,E2 -19651.982} C_VEL
LIN {X 0,Y 236.349,Z 368.722,A -85,B 0,C 180,E1 -19653.9,E2 -19653.9} C_VEL
LIN {X 0,Y 237.244,Z 358.264,A -85,B 0,C 180,E1 -19655.545,E2 -19655.545} C_VEL
LIN {X 0,Y 238.161,Z 345.721,A -85,B 0,C 180,E1 -19657.064,E2 -19657.064} C_VEL
LIN {X 0,Y 238.835,Z 333.321,A -85,B 0,C 180,E1 -19658.165,E2 -19658.165} C_VEL
LIN {X 0,Y 239.297,Z 320.42,A -85,B 0,C 180,E1 -19658.952,E2 -19658.952} C_VEL
LIN {X 0,Y 241.312,Z 261.059,A -85,B 0,C 180,E1 -19661.492,E2 -19661.492} C_VEL
LIN {X 0,Y 238.22,Z 235.353,A -85,B 0,C 180,E1 -19662.826,E2 -19662.826} C_VEL
LIN {X 0,Y 238.254,Z 232.134,A -85,B 0,C 180,E1 -19663.8,E2 -19663.8} C_VEL
LIN {X 0,Y 236.159,Z 220.985,A -85,B 0,C 180,E1 -19667.672,E2 -19667.672} C_VEL
LIN {X 0,Y 235.051,Z 215.426,A -85,B 0,C 180,E1 -19669.715,E2 -19669.715} C_VEL
LIN {X 0,Y 234.938,Z 215.221,A -85,B 0,C 180,E1 -19673.869,E2 -19673.869} C_VEL
LIN {X 0,Y 234.958,Z 215.219,A -85,B 0,C 180,E1 -19677.423,E2 -19677.423} C_VEL
LIN {X 0,Y 234.952,Z 215.22,A -85,B 0,C 180,E1 -19681.405,E2 -19681.405} C_VEL
LIN {X 0,Y 234.987,Z 215.214,A -85,B 0,C 180,E1 -19685.246,E2 -19685.246} C_VEL
LIN {X 0,Y 235.01,Z 215.21,A -85,B 0,C 180,E1 -19688.969,E2 -19688.969} C_VEL
LIN {X 0,Y 235.095,Z 215.2,A -85,B 0,C 180,E1 -19693.058,E2 -19693.058} C_VEL
LIN {X 0,Y 235.145,Z 215.192,A -85,B 0,C 180,E1 -19697.923,E2 -19697.923} C_VEL
LIN {X 0,Y 235.389,Z 215.163,A -85,B 0,C 180,E1 -19701.413,E2 -19701.413} C_VEL
LIN {X 0,Y 235.404,Z 215.162,A -85,B 0,C 180,E1 -19703.14,E2 -19703.14} C_VEL
LIN {X 0,Y 235.594,Z 215.135,A -85,B 0,C 180,E1 -19708.289,E2 -19708.289} C_VEL
LIN {X 0,Y 235.594,Z 215.136,A -85,B 0,C 180,E1 -19711.708,E2 -19711.708} C_VEL
LIN {X 0,Y 235.399,Z 215.163,A -85,B 0,C 180,E1 -19716.857,E2 -19716.857} C_VEL
LIN {X 0,Y 235.234,Z 215.181,A -85,B 0,C 180,E1 -19720.325,E2 -19720.325} C_VEL
LIN {X 0,Y 235.11,Z 215.195,A -85,B 0,C 180,E1 -19725.605,E2 -19725.605} C_VEL
LIN {X 0,Y 235.004,Z 215.211,A -85,B 0,C 180,E1 -19729.204,E2 -19729.204} C_VEL
LIN {X 0,Y 234.956,Z 215.217,A -85,B 0,C 180,E1 -19732.882,E2 -19732.882} C_VEL
LIN {X 0,Y 234.965,Z 215.217,A -85,B 0,C 180,E1 -19736.656,E2 -19736.656} C_VEL
LIN {X 0,Y 234.927,Z 215.223,A -85,B 0,C 180,E1 -19740.567,E2 -19740.567} C_VEL
LIN {X 0,Y 234.955,Z 215.218,A -85,B 0,C 180,E1 -19744.632,E2 -19744.632} C_VEL
LIN {X 0,Y 234.96,Z 215.216,A -85,B 0,C 180,E1 -19748.951,E2 -19748.951} C_VEL
LIN {X 0,Y 234.959,Z 215.214,A -85,B 0,C 180,E1 -19753.467,E2 -19753.467} C_VEL
LIN {X 0,Y 234.954,Z 215.219,A -85,B 0,C 180,E1 -19756.531,E2 -19756.531} C_VEL
LIN {X 0,Y 234.948,Z 215.215,A -85,B 0,C 180,E1 -19761.086,E2 -19761.086} C_VEL
LIN {X 0,Y 234.954,Z 215.216,A -85,B 0,C 180,E1 -19765.367,E2 -19765.367} C_VEL
LIN {X 0,Y 234.961,Z 215.217,A -85,B 0,C 180,E1 -19770.158,E2 -19770.158} C_VEL
LIN {X 0,Y 234.987,Z 215.214,A -85,B 0,C 180,E1 -19773.794,E2 -19773.794} C_VEL
LIN {X 0,Y 235.004,Z 215.209,A -85,B 0,C 180,E1 -19778.97,E2 -19778.97} C_VEL
LIN {X 0,Y 235.089,Z 215.199,A -85,B 0,C 180,E1 -19783.06,E2 -19783.06} C_VEL
LIN {X 0,Y 235.108,Z 215.201,A -85,B 0,C 180,E1 -19787.923,E2 -19787.923} C_VEL
LIN {X 0,Y 235.324,Z 215.171,A -85,B 0,C 180,E1 -19791.413,E2 -19791.413} C_VEL
LIN {X 0,Y 235.367,Z 215.163,A -85,B 0,C 180,E1 -19793.141,E2 -19793.141} C_VEL
LIN {X 0,Y 235.589,Z 215.138,A -85,B 0,C 180,E1 -19798.291,E2 -19798.291} C_VEL
LIN {X 0,Y 235.589,Z 215.138,A -85,B 0,C 180,E1 -19801.71,E2 -19801.71} C_VEL
LIN {X 0,Y 235.398,Z 215.161,A -85,B 0,C 180,E1 -19806.86,E2 -19806.86} C_VEL
LIN {X 0,Y 235.232,Z 215.178,A -85,B 0,C 180,E1 -19810.328,E2 -19810.328} C_VEL
LIN {X 0,Y 235.108,Z 215.199,A -85,B 0,C 180,E1 -19815.608,E2 -19815.608} C_VEL
LIN {X 0,Y 235.004,Z 215.21,A -85,B 0,C 180,E1 -19819.207,E2 -19819.207} C_VEL
LIN {X 0,Y 234.956,Z 215.217,A -85,B 0,C 180,E1 -19822.884,E2 -19822.884} C_VEL
LIN {X 0,Y 234.963,Z 215.214,A -85,B 0,C 180,E1 -19826.659,E2 -19826.659} C_VEL
LIN {X 0,Y 234.9,Z 215.22,A -85,B 0,C 180,E1 -19831.058,E2 -19831.058} C_VEL
LIN {X 0,Y 234.923,Z 215.221,A -85,B 0,C 180,E1 -19834.64,E2 -19834.64} C_VEL
LIN {X 0,Y 234.89,Z 215.223,A -85,B 0,C 180,E1 -19838.489,E2 -19838.489} C_VEL
LIN {X 0,Y 234.266,Z 215.308,A -85,B 0,C 180,E1 -19839.919,E2 -19839.919} C_VEL
LIN {X 0,Y 231.405,Z 215.666,A -85,B 0,C 180,E1 -19842.251,E2 -19842.251} C_VEL
LIN {X 0,Y 228.937,Z 215.968,A -85,B 0,C 180,E1 -19844.152,E2 -19844.152} C_VEL
LIN {X 0,Y 227.868,Z 216.101,A -85,B 0,C 180,E1 -19845.629,E2 -19845.629} C_VEL
LIN {X 0,Y 227.778,Z 216.109,A -85,B 0,C 180,E1 -19846.13,E2 -19846.13} C_VEL
LIN {X 0,Y 227.934,Z 216.262,A -85,B 0,C 180,E1 -19851.363,E2 -19851.363} C_VEL
LIN {X 0,Y 230.666,Z 228.402,A -85,B 0,C 180,E1 -19855.352,E2 -19855.352} C_VEL
LIN {X 0,Y 233.606,Z 242.159,A -85,B 0,C 180,E1 -19859.605,E2 -19859.605} C_VEL
LIN {X 0,Y 233.945,Z 246.014,A -85,B 0,C 180,E1 -19860.731,E2 -19860.731} C_VEL
LIN {X 0,Y 232.155,Z 255.932,A -85,B 0,C 180,E1 -19863.429,E2 -19863.429} C_VEL
LIN {X 0,Y 233.175,Z 278.937,A -85,B 0,C 180,E1 -19864.481,E2 -19864.481} C_VEL
LIN {X 0,Y 234.75,Z 301.958,A -85,B 0,C 180,E1 -19865.516,E2 -19865.516} C_VEL
LIN {X 0,Y 232.956,Z 358.354,A -85,B 0,C 180,E1 -19867.788,E2 -19867.788} C_VEL
LIN {X 0,Y 232.252,Z 370.631,A -85,B 0,C 180,E1 -19868.593,E2 -19868.593} C_VEL
LIN {X 0,Y 231.45,Z 381.257,A -85,B 0,C 180,E1 -19869.563,E2 -19869.563} C_VEL
LIN {X 0,Y 230.271,Z 393.224,A -85,B 0,C 180,E1 -19871.014,E2 -19871.014} C_VEL
LIN {X 0,Y 229.137,Z 404.784,A -85,B 0,C 180,E1 -19872.831,E2 -19872.831} C_VEL
LIN {X 0,Y 228.059,Z 414.681,A -85,B 0,C 180,E1 -19874.816,E2 -19874.816} C_VEL
LIN {X 0,Y 227.318,Z 423.661,A -85,B 0,C 180,E1 -19877.049,E2 -19877.049} C_VEL
LIN {X 0,Y 226.884,Z 430.97,A -85,B 0,C 180,E1 -19879.29,E2 -19879.29} C_VEL
LIN {X 0,Y 226.701,Z 437.962,A -85,B 0,C 180,E1 -19881.983,E2 -19881.983} C_VEL
LIN {X 0,Y 226.81,Z 443.409,A -85,B 0,C 180,E1 -19884.667,E2 -19884.667} C_VEL
LIN {X 0,Y 226.961,Z 447.47,A -85,B 0,C 180,E1 -19887.339,E2 -19887.339} C_VEL
LIN {X 0,Y 227.057,Z 450.282,A -85,B 0,C 180,E1 -19890.001,E2 -19890.001} C_VEL
LIN {X 0,Y 226.892,Z 451.482,A -85,B 0,C 180,E1 -19891.776,E2 -19891.776} C_VEL
LIN {X 0,Y 226.514,Z 452.197,A -85,B 0,C 180,E1 -19893.559,E2 -19893.559} C_VEL
LIN {X 0,Y 226.157,Z 452.488,A -85,B 0,C 180,E1 -19896.046,E2 -19896.046} C_VEL
LIN {X 0,Y 226.094,Z 451.805,A -85,B 0,C 180,E1 -19898.942,E2 -19898.942} C_VEL
LIN {X 0,Y 226.759,Z 449.516,A -85,B 0,C 180,E1 -19902.531,E2 -19902.531} C_VEL
LIN {X 0,Y 228.068,Z 446.695,A -85,B 0,C 180,E1 -19905.186,E2 -19905.186} C_VEL
LIN {X 0,Y 229.854,Z 442.869,A -85,B 0,C 180,E1 -19907.805,E2 -19907.805} C_VEL
LIN {X 0,Y 232.518,Z 437.135,A -85,B 0,C 180,E1 -19910.757,E2 -19910.757} C_VEL
LIN {X 0,Y 235.53,Z 430.711,A -85,B 0,C 180,E1 -19913.29,E2 -19913.29} C_VEL
LIN {X 0,Y 239.23,Z 422.886,A -85,B 0,C 180,E1 -19915.679,E2 -19915.679} C_VEL
LIN {X 0,Y 243.372,Z 413.227,A -85,B 0,C 180,E1 -19917.987,E2 -19917.987} C_VEL
LIN {X 0,Y 247.256,Z 403.357,A -85,B 0,C 180,E1 -19919.83,E2 -19919.83} C_VEL
LIN {X 0,Y 251.078,Z 392.318,A -85,B 0,C 180,E1 -19921.423,E2 -19921.423} C_VEL
LIN {X 0,Y 254.846,Z 379.883,A -85,B 0,C 180,E1 -19922.767,E2 -19922.767} C_VEL
LIN {X 0,Y 258.016,Z 366.704,A -85,B 0,C 180,E1 -19923.828,E2 -19923.828} C_VEL
LIN {X 0,Y 260.38,Z 353.003,A -85,B 0,C 180,E1 -19924.615,E2 -19924.615} C_VEL
LIN {X 0,Y 265.053,Z 308.913,A -85,B 0,C 180,E1 -19926.353,E2 -19926.353} C_VEL
LIN {X 0,Y 264.816,Z 295.766,A -85,B 0,C 180,E1 -19927.38,E2 -19927.38} C_VEL
LIN {X 0,Y 264.214,Z 285.654,A -85,B 0,C 180,E1 -19928.371,E2 -19928.371} C_VEL
LIN {X 0,Y 261.35,Z 278.505,A -85,B 0,C 180,E1 -19930.004,E2 -19930.004} C_VEL
LIN {X 0,Y 258.559,Z 272.73,A -85,B 0,C 180,E1 -19931.72,E2 -19931.72} C_VEL
LIN {X 0,Y 255.697,Z 267.471,A -85,B 0,C 180,E1 -19933.673,E2 -19933.673} C_VEL
LIN {X 0,Y 252.332,Z 261.415,A -85,B 0,C 180,E1 -19936.49,E2 -19936.49} C_VEL
LIN {X 0,Y 249.263,Z 256.662,A -85,B 0,C 180,E1 -19939.979,E2 -19939.979} C_VEL
LIN {X 0,Y 247.845,Z 254.028,A -85,B 0,C 180,E1 -19942.671,E2 -19942.671} C_VEL
LIN {X 0,Y 247.132,Z 252.651,A -85,B 0,C 180,E1 -19945.335,E2 -19945.335} C_VEL
LIN {X 0,Y 247.342,Z 252.448,A -85,B 0,C 180,E1 -19949.238,E2 -19949.238} C_VEL
LIN {X 0,Y 248.815,Z 254.115,A -85,B 0,C 180,E1 -19952.694,E2 -19952.694} C_VEL
LIN {X 0,Y 251.289,Z 256.877,A -85,B 0,C 180,E1 -19955.828,E2 -19955.828} C_VEL
LIN {X 0,Y 255.022,Z 261.991,A -85,B 0,C 180,E1 -19959.168,E2 -19959.168} C_VEL
LIN {X 0,Y 258.274,Z 267.01,A -85,B 0,C 180,E1 -19961.481,E2 -19961.481} C_VEL
LIN {X 0,Y 261.152,Z 271.983,A -85,B 0,C 180,E1 -19963.26,E2 -19963.26} C_VEL
LIN {X 0,Y 263.447,Z 276.257,A -85,B 0,C 180,E1 -19964.56,E2 -19964.56} C_VEL
LIN {X 0,Y 266.377,Z 282.451,A -85,B 0,C 180,E1 -19966.126,E2 -19966.126} C_VEL
LIN {X 0,Y 266.956,Z 284.146,A -85,B 0,C 180,E1 -19966.463,E2 -19966.463} C_VEL
LIN {X 0,Y 261.504,Z 329.882,A -85,B 0,C 180,E1 -19968.469,E2 -19968.469} C_VEL
LIN {X 0,Y 259.648,Z 342.525,A -85,B 0,C 180,E1 -19969.305,E2 -19969.305} C_VEL
LIN {X 0,Y 257.254,Z 354.364,A -85,B 0,C 180,E1 -19970.393,E2 -19970.393} C_VEL
LIN {X 0,Y 254.582,Z 364.647,A -85,B 0,C 180,E1 -19971.626,E2 -19971.626} C_VEL
LIN {X 0,Y 251.427,Z 374.806,A -85,B 0,C 180,E1 -19973.177,E2 -19973.177} C_VEL
LIN {X 0,Y 248.529,Z 382.868,A -85,B 0,C 180,E1 -19974.726,E2 -19974.726} C_VEL
LIN {X 0,Y 245.045,Z 391.118,A -85,B 0,C 180,E1 -19976.711,E2 -19976.711} C_VEL
LIN {X 0,Y 241.904,Z 397.683,A -85,B 0,C 180,E1 -19978.751,E2 -19978.751} C_VEL
LIN {X 0,Y 238.98,Z 403.045,A -85,B 0,C 180,E1 -19980.847,E2 -19980.847} C_VEL
LIN {X 0,Y 235.914,Z 407.936,A -85,B 0,C 180,E1 -19983.415,E2 -19983.415} C_VEL
LIN {X 0,Y 233.232,Z 411.437,A -85,B 0,C 180,E1 -19986.066,E2 -19986.066} C_VEL
LIN {X 0,Y 231.09,Z 413.585,A -85,B 0,C 180,E1 -19988.746,E2 -19988.746} C_VEL
LIN {X 0,Y 229.4,Z 414.496,A -85,B 0,C 180,E1 -19991.369,E2 -19991.369} C_VEL
LIN {X 0,Y 227.976,Z 414.214,A -85,B 0,C 180,E1 -19994.277,E2 -19994.277} C_VEL
LIN {X 0,Y 227.211,Z 413.094,A -85,B 0,C 180,E1 -19996.486,E2 -19996.486} C_VEL
LIN {X 0,Y 226.657,Z 410.889,A -85,B 0,C 180,E1 -19999,E2 -19999} C_VEL
LIN {X 0,Y 226.447,Z 407.073,A -85,B 0,C 180,E1 -20001.865,E2 -20001.865} C_VEL
LIN {X 0,Y 226.641,Z 401.688,A -85,B 0,C 180,E1 -20004.747,E2 -20004.747} C_VEL
LIN {X 0,Y 227.047,Z 395.648,A -85,B 0,C 180,E1 -20007.206,E2 -20007.206} C_VEL
LIN {X 0,Y 227.599,Z 388.247,A -85,B 0,C 180,E1 -20009.607,E2 -20009.607} C_VEL
LIN {X 0,Y 228.324,Z 379.729,A -85,B 0,C 180,E1 -20011.81,E2 -20011.81} C_VEL
LIN {X 0,Y 229.191,Z 369.941,A -85,B 0,C 180,E1 -20013.845,E2 -20013.845} C_VEL
LIN {X 0,Y 230.203,Z 358.432,A -85,B 0,C 180,E1 -20015.723,E2 -20015.723} C_VEL
LIN {X 0,Y 231.152,Z 345.581,A -85,B 0,C 180,E1 -20017.313,E2 -20017.313} C_VEL
LIN {X 0,Y 231.918,Z 332.028,A -85,B 0,C 180,E1 -20018.514,E2 -20018.514} C_VEL
LIN {X 0,Y 232.346,Z 318.315,A -85,B 0,C 180,E1 -20019.315,E2 -20019.315} C_VEL
LIN {X 0,Y 234.393,Z 262.018,A -85,B 0,C 180,E1 -20021.789,E2 -20021.789} C_VEL
LIN {X 0,Y 231.268,Z 235.606,A -85,B 0,C 180,E1 -20023.208,E2 -20023.208} C_VEL
LIN {X 0,Y 231.083,Z 231.901,A -85,B 0,C 180,E1 -20024.386,E2 -20024.386} C_VEL
LIN {X 0,Y 229.013,Z 221.493,A -85,B 0,C 180,E1 -20028.127,E2 -20028.127} C_VEL
LIN {X 0,Y 227.967,Z 216.258,A -85,B 0,C 180,E1 -20030.123,E2 -20030.123} C_VEL
LIN {X 0,Y 227.883,Z 216.099,A -85,B 0,C 180,E1 -20034.128,E2 -20034.128} C_VEL
LIN {X 0,Y 227.871,Z 216.099,A -85,B 0,C 180,E1 -20038.377,E2 -20038.377} C_VEL
LIN {X 0,Y 227.886,Z 216.097,A -85,B 0,C 180,E1 -20042.444,E2 -20042.444} C_VEL
LIN {X 0,Y 227.913,Z 216.093,A -85,B 0,C 180,E1 -20046.366,E2 -20046.366} C_VEL
LIN {X 0,Y 227.942,Z 216.09,A -85,B 0,C 180,E1 -20050.173,E2 -20050.173} C_VEL
LIN {X 0,Y 228.056,Z 216.075,A -85,B 0,C 180,E1 -20053.897,E2 -20053.897} C_VEL
LIN {X 0,Y 228.17,Z 216.063,A -85,B 0,C 180,E1 -20059.349,E2 -20059.349} C_VEL
LIN {X 0,Y 228.356,Z 216.038,A -85,B 0,C 180,E1 -20062.927,E2 -20062.927} C_VEL
LIN {X 0,Y 228.553,Z 216.012,A -85,B 0,C 180,E1 -20068.237,E2 -20068.237} C_VEL
LIN {X 0,Y 228.552,Z 216.013,A -85,B 0,C 180,E1 -20071.761,E2 -20071.761} C_VEL
LIN {X 0,Y 228.351,Z 216.039,A -85,B 0,C 180,E1 -20077.07,E2 -20077.07} C_VEL
LIN {X 0,Y 228.16,Z 216.064,A -85,B 0,C 180,E1 -20080.649,E2 -20080.649} C_VEL
LIN {X 0,Y 228.061,Z 216.075,A -85,B 0,C 180,E1 -20084.271,E2 -20084.271} C_VEL
LIN {X 0,Y 227.999,Z 216.081,A -85,B 0,C 180,E1 -20087.952,E2 -20087.952} C_VEL
LIN {X 0,Y 227.926,Z 216.093,A -85,B 0,C 180,E1 -20092.328,E2 -20092.328} C_VEL
LIN {X 0,Y 227.938,Z 216.092,A -85,B 0,C 180,E1 -20096.602,E2 -20096.602} C_VEL
LIN {X 0,Y 227.903,Z 216.096,A -85,B 0,C 180,E1 -20100.295,E2 -20100.295} C_VEL
LIN {X 0,Y 227.884,Z 216.094,A -85,B 0,C 180,E1 -20103.717,E2 -20103.717} C_VEL
LIN {X 0,Y 227.865,Z 216.101,A -85,B 0,C 180,E1 -20108.085,E2 -20108.085} C_VEL
LIN {X 0,Y 227.903,Z 216.095,A -85,B 0,C 180,E1 -20112.719,E2 -20112.719} C_VEL
LIN {X 0,Y 227.891,Z 216.096,A -85,B 0,C 180,E1 -20117.741,E2 -20117.741} C_VEL
LIN {X 0,Y 227.864,Z 216.099,A -85,B 0,C 180,E1 -20121.914,E2 -20121.914} C_VEL
LIN {X 0,Y 227.884,Z 216.098,A -85,B 0,C 180,E1 -20126.373,E2 -20126.373} C_VEL
LIN {X 0,Y 227.911,Z 216.095,A -85,B 0,C 180,E1 -20130.438,E2 -20130.438} C_VEL
LIN {X 0,Y 227.921,Z 216.093,A -85,B 0,C 180,E1 -20134.426,E2 -20134.426} C_VEL
LIN {X 0,Y 227.955,Z 216.089,A -85,B 0,C 180,E1 -20138.287,E2 -20138.287} C_VEL
LIN {X 0,Y 228.028,Z 216.078,A -85,B 0,C 180,E1 -20142.826,E2 -20142.826} C_VEL
LIN {X 0,Y 228.066,Z 216.075,A -85,B 0,C 180,E1 -20147.544,E2 -20147.544} C_VEL
LIN {X 0,Y 228.26,Z 216.05,A -85,B 0,C 180,E1 -20151.145,E2 -20151.145} C_VEL
LIN {X 0,Y 228.317,Z 216.041,A -85,B 0,C 180,E1 -20152.928,E2 -20152.928} C_VEL
LIN {X 0,Y 228.547,Z 216.015,A -85,B 0,C 180,E1 -20158.239,E2 -20158.239} C_VEL
LIN {X 0,Y 228.548,Z 216.014,A -85,B 0,C 180,E1 -20161.763,E2 -20161.763} C_VEL
LIN {X 0,Y 228.349,Z 216.04,A -85,B 0,C 180,E1 -20167.072,E2 -20167.072} C_VEL
LIN {X 0,Y 228.153,Z 216.06,A -85,B 0,C 180,E1 -20170.652,E2 -20170.652} C_VEL
LIN {X 0,Y 228.059,Z 216.075,A -85,B 0,C 180,E1 -20174.273,E2 -20174.273} C_VEL
LIN {X 0,Y 227.998,Z 216.081,A -85,B 0,C 180,E1 -20177.955,E2 -20177.955} C_VEL
LIN {X 0,Y 227.926,Z 216.092,A -85,B 0,C 180,E1 -20182.331,E2 -20182.331} C_VEL
LIN {X 0,Y 227.938,Z 216.089,A -85,B 0,C 180,E1 -20186.604,E2 -20186.604} C_VEL
LIN {X 0,Y 227.893,Z 216.096,A -85,B 0,C 180,E1 -20190.292,E2 -20190.292} C_VEL
LIN {X 0,Y 227.873,Z 216.099,A -85,B 0,C 180,E1 -20193.722,E2 -20193.722} C_VEL
LIN {X 0,Y 227.84,Z 216.102,A -85,B 0,C 180,E1 -20198.093,E2 -20198.093} C_VEL
LIN {X 0,Y 227.803,Z 216.11,A -85,B 0,C 180,E1 -20202.745,E2 -20202.745} C_VEL
LIN {X 0,Y 227.778,Z 216.109,A -85,B 0,C 180,E1 -20206.13,E2 -20206.13} C_VEL
LIN {X 0,Y 227.024,Z 216.268,A -85,B 0,C 180,E1 -20207.164,E2 -20207.164} C_VEL
LIN {X 0,Y 221.366,Z 216.969,A -85,B 0,C 180,E1 -20210.366,E2 -20210.366} C_VEL
LIN {X 0,Y 221.011,Z 217.744,A -85,B 0,C 180,E1 -20211.135,E2 -20211.135} C_VEL
LIN {X 0,Y 221.078,Z 218.064,A -85,B 0,C 180,E1 -20211.269,E2 -20211.269} C_VEL
LIN {X 0,Y 223.664,Z 229.63,A -85,B 0,C 180,E1 -20215.152,E2 -20215.152} C_VEL
LIN {X 0,Y 226.397,Z 242.28,A -85,B 0,C 180,E1 -20219.192,E2 -20219.192} C_VEL
LIN {X 0,Y 227.023,Z 245.922,A -85,B 0,C 180,E1 -20220.311,E2 -20220.311} C_VEL
LIN {X 0,Y 225.248,Z 255.644,A -85,B 0,C 180,E1 -20223.031,E2 -20223.031} C_VEL
LIN {X 0,Y 225.961,Z 275.222,A -85,B 0,C 180,E1 -20223.962,E2 -20223.962} C_VEL
LIN {X 0,Y 227.77,Z 302.412,A -85,B 0,C 180,E1 -20225.22,E2 -20225.22} C_VEL
LIN {X 0,Y 225.944,Z 357.739,A -85,B 0,C 180,E1 -20227.543,E2 -20227.543} C_VEL
LIN {X 0,Y 225.252,Z 369.983,A -85,B 0,C 180,E1 -20228.375,E2 -20228.375} C_VEL
LIN {X 0,Y 224.409,Z 380.554,A -85,B 0,C 180,E1 -20229.372,E2 -20229.372} C_VEL
LIN {X 0,Y 223.284,Z 391.934,A -85,B 0,C 180,E1 -20230.784,E2 -20230.784} C_VEL
LIN {X 0,Y 222.087,Z 404.066,A -85,B 0,C 180,E1 -20232.744,E2 -20232.744} C_VEL
LIN {X 0,Y 221.01,Z 413.958,A -85,B 0,C 180,E1 -20234.792,E2 -20234.792} C_VEL
LIN {X 0,Y 220.258,Z 422.933,A -85,B 0,C 180,E1 -20237.095,E2 -20237.095} C_VEL
LIN {X 0,Y 219.847,Z 430.261,A -85,B 0,C 180,E1 -20239.409,E2 -20239.409} C_VEL
LIN {X 0,Y 219.673,Z 437.255,A -85,B 0,C 180,E1 -20242.187,E2 -20242.187} C_VEL
LIN {X 0,Y 219.781,Z 441.898,A -85,B 0,C 180,E1 -20244.496,E2 -20244.496} C_VEL
LIN {X 0,Y 219.958,Z 446.159,A -85,B 0,C 180,E1 -20247.254,E2 -20247.254} C_VEL
LIN {X 0,Y 220.038,Z 449.145,A -85,B 0,C 180,E1 -20250.001,E2 -20250.001} C_VEL
LIN {X 0,Y 219.842,Z 450.483,A -85,B 0,C 180,E1 -20251.833,E2 -20251.833} C_VEL
LIN {X 0,Y 219.46,Z 451.29,A -85,B 0,C 180,E1 -20253.673,E2 -20253.673} C_VEL
LIN {X 0,Y 219.102,Z 451.713,A -85,B 0,C 180,E1 -20256.077,E2 -20256.077} C_VEL
LIN {X 0,Y 219.049,Z 451.212,A -85,B 0,C 180,E1 -20259.233,E2 -20259.233} C_VEL
LIN {X 0,Y 219.789,Z 449.093,A -85,B 0,C 180,E1 -20262.935,E2 -20262.935} C_VEL
LIN {X 0,Y 221.186,Z 446.463,A -85,B 0,C 180,E1 -20265.67,E2 -20265.67} C_VEL
LIN {X 0,Y 223.1,Z 442.856,A -85,B 0,C 180,E1 -20268.363,E2 -20268.363} C_VEL
LIN {X 0,Y 225.397,Z 438.354,A -85,B 0,C 180,E1 -20270.918,E2 -20270.918} C_VEL
LIN {X 0,Y 228.499,Z 432.328,A -85,B 0,C 180,E1 -20273.57,E2 -20273.57} C_VEL
LIN {X 0,Y 232.24,Z 425.138,A -85,B 0,C 180,E1 -20276.028,E2 -20276.028} C_VEL
LIN {X 0,Y 236.475,Z 416.221,A -85,B 0,C 180,E1 -20278.394,E2 -20278.394} C_VEL
LIN {X 0,Y 240.374,Z 407.165,A -85,B 0,C 180,E1 -20280.289,E2 -20280.289} C_VEL
LIN {X 0,Y 244.705,Z 396.006,A -85,B 0,C 180,E1 -20282.096,E2 -20282.096} C_VEL
LIN {X 0,Y 248.57,Z 384.942,A -85,B 0,C 180,E1 -20283.46,E2 -20283.46} C_VEL
LIN {X 0,Y 252.05,Z 372.569,A -85,B 0,C 180,E1 -20284.62,E2 -20284.62} C_VEL
LIN {X 0,Y 254.893,Z 359.667,A -85,B 0,C 180,E1 -20285.504,E2 -20285.504} C_VEL
LIN {X 0,Y 256.932,Z 346.17,A -85,B 0,C 180,E1 -20286.144,E2 -20286.144} C_VEL
LIN {X 0,Y 260.876,Z 310.149,A -85,B 0,C 180,E1 -20287.58,E2 -20287.58} C_VEL
LIN {X 0,Y 260.825,Z 297.879,A -85,B 0,C 180,E1 -20288.574,E2 -20288.574} C_VEL
LIN {X 0,Y 260.418,Z 289.604,A -85,B 0,C 180,E1 -20289.399,E2 -20289.399} C_VEL
LIN {X 0,Y 257.787,Z 282.807,A -85,B 0,C 180,E1 -20291.082,E2 -20291.082} C_VEL
LIN {X 0,Y 255.603,Z 278.186,A -85,B 0,C 180,E1 -20292.52,E2 -20292.52} C_VEL
LIN {X 0,Y 253.183,Z 273.403,A -85,B 0,C 180,E1 -20294.354,E2 -20294.354} C_VEL
LIN {X 0,Y 250.237,Z 267.799,A -85,B 0,C 180,E1 -20297.03,E2 -20297.03} C_VEL
LIN {X 0,Y 247.497,Z 263.297,A -85,B 0,C 180,E1 -20300.385,E2 -20300.385} C_VEL
LIN {X 0,Y 246.186,Z 260.68,A -85,B 0,C 180,E1 -20303.165,E2 -20303.165} C_VEL
LIN {X 0,Y 245.639,Z 259.532,A -85,B 0,C 180,E1 -20305.607,E2 -20305.607} C_VEL
LIN {X 0,Y 245.938,Z 259.467,A -85,B 0,C 180,E1 -20309.52,E2 -20309.52} C_VEL
LIN {X 0,Y 247.589,Z 261.358,A -85,B 0,C 180,E1 -20313.111,E2 -20313.111} C_VEL
LIN {X 0,Y 249.546,Z 263.777,A -85,B 0,C 180,E1 -20315.649,E2 -20315.649} C_VEL
LIN {X 0,Y 252.825,Z 268.508,A -85,B 0,C 180,E1 -20318.748,E2 -20318.748} C_VEL
LIN {X 0,Y 255.717,Z 273.183,A -85,B 0,C 180,E1 -20320.939,E2 -20320.939} C_VEL
LIN {X 0,Y 259.149,Z 279.322,A -85,B 0,C 180,E1 -20323.16,E2 -20323.16} C_VEL
LIN {X 0,Y 262.486,Z 286.54,A -85,B 0,C 180,E1 -20325.133,E2 -20325.133} C_VEL
LIN {X 0,Y 262.705,Z 287.549,A -85,B 0,C 180,E1 -20325.301,E2 -20325.301} C_VEL
LIN {X 0,Y 257.209,Z 330.868,A -85,B 0,C 180,E1 -20327.243,E2 -20327.243} C_VEL
LIN {X 0,Y 255.046,Z 344.402,A -85,B 0,C 180,E1 -20328.173,E2 -20328.173} C_VEL
LIN {X 0,Y 252.568,Z 355.755,A -85,B 0,C 180,E1 -20329.244,E2 -20329.244} C_VEL
LIN {X 0,Y 249.543,Z 366.653,A -85,B 0,C 180,E1 -20330.582,E2 -20330.582} C_VEL
LIN {X 0,Y 246.078,Z 376.809,A -85,B 0,C 180,E1 -20332.202,E2 -20332.202} C_VEL
LIN {X 0,Y 243,Z 384.605,A -85,B 0,C 180,E1 -20333.773,E2 -20333.773} C_VEL
LIN {X 0,Y 239.16,Z 392.976,A -85,B 0,C 180,E1 -20335.884,E2 -20335.884} C_VEL
LIN {X 0,Y 235.99,Z 399.11,A -85,B 0,C 180,E1 -20337.866,E2 -20337.866} C_VEL
LIN {X 0,Y 232.895,Z 404.298,A -85,B 0,C 180,E1 -20339.999,E2 -20339.999} C_VEL
LIN {X 0,Y 229.597,Z 409.028,A -85,B 0,C 180,E1 -20342.631,E2 -20342.631} C_VEL
LIN {X 0,Y 226.754,Z 412.433,A -85,B 0,C 180,E1 -20345.334,E2 -20345.334} C_VEL
LIN {X 0,Y 225.161,Z 413.924,A -85,B 0,C 180,E1 -20347.171,E2 -20347.171} C_VEL
LIN {X 0,Y 223.769,Z 414.901,A -85,B 0,C 180,E1 -20349.034,E2 -20349.034} C_VEL
LIN {X 0,Y 222.262,Z 415.341,A -85,B 0,C 180,E1 -20351.408,E2 -20351.408} C_VEL
LIN {X 0,Y 221.531,Z 415.195,A -85,B 0,C 180,E1 -20352.83,E2 -20352.83} C_VEL
LIN {X 0,Y 220.675,Z 414.509,A -85,B 0,C 180,E1 -20354.76,E2 -20354.76} C_VEL
LIN {X 0,Y 220.043,Z 413.272,A -85,B 0,C 180,E1 -20356.705,E2 -20356.705} C_VEL
LIN {X 0,Y 219.509,Z 410.315,A -85,B 0,C 180,E1 -20359.643,E2 -20359.643} C_VEL
LIN {X 0,Y 219.371,Z 405.929,A -85,B 0,C 180,E1 -20362.608,E2 -20362.608} C_VEL
LIN {X 0,Y 219.647,Z 400.041,A -85,B 0,C 180,E1 -20365.535,E2 -20365.535} C_VEL
LIN {X 0,Y 220.118,Z 393.303,A -85,B 0,C 180,E1 -20368.094,E2 -20368.094} C_VEL
LIN {X 0,Y 220.793,Z 384.955,A -85,B 0,C 180,E1 -20370.616,E2 -20370.616} C_VEL
LIN {X 0,Y 221.63,Z 375.437,A -85,B 0,C 180,E1 -20372.89,E2 -20372.89} C_VEL
LIN {X 0,Y 222.539,Z 365.377,A -85,B 0,C 180,E1 -20374.803,E2 -20374.803} C_VEL
LIN {X 0,Y 223.488,Z 353.817,A -85,B 0,C 180,E1 -20376.535,E2 -20376.535} C_VEL
LIN {X 0,Y 224.379,Z 341.581,A -85,B 0,C 180,E1 -20377.929,E2 -20377.929} C_VEL
LIN {X 0,Y 225.074,Z 327.852,A -85,B 0,C 180,E1 -20379.04,E2 -20379.04} C_VEL
LIN {X 0,Y 225.683,Z 306.663,A -85,B 0,C 180,E1 -20380.107,E2 -20380.107} C_VEL
LIN {X 0,Y 227.415,Z 262.532,A -85,B 0,C 180,E1 -20382.123,E2 -20382.123} C_VEL
LIN {X 0,Y 224.294,Z 235.803,A -85,B 0,C 180,E1 -20383.61,E2 -20383.61} C_VEL
LIN {X 0,Y 223.789,Z 231.63,A -85,B 0,C 180,E1 -20385.04,E2 -20385.04} C_VEL
LIN {X 0,Y 221.804,Z 221.625,A -85,B 0,C 180,E1 -20388.738,E2 -20388.738} C_VEL
LIN {X 0,Y 220.905,Z 217.176,A -85,B 0,C 180,E1 -20390.483,E2 -20390.483} C_VEL
LIN {X 0,Y 220.803,Z 216.981,A -85,B 0,C 180,E1 -20395.044,E2 -20395.044} C_VEL
LIN {X 0,Y 220.868,Z 216.974,A -85,B 0,C 180,E1 -20399.394,E2 -20399.394} C_VEL
LIN {X 0,Y 220.895,Z 216.97,A -85,B 0,C 180,E1 -20403.548,E2 -20403.548} C_VEL
LIN {X 0,Y 220.877,Z 216.972,A -85,B 0,C 180,E1 -20407.552,E2 -20407.552} C_VEL
LIN {X 0,Y 220.983,Z 216.955,A -85,B 0,C 180,E1 -20412.57,E2 -20412.57} C_VEL
LIN {X 0,Y 221.025,Z 216.954,A -85,B 0,C 180,E1 -20417.138,E2 -20417.138} C_VEL
LIN {X 0,Y 221.256,Z 216.922,A -85,B 0,C 180,E1 -20420.86,E2 -20420.86} C_VEL
LIN {X 0,Y 221.294,Z 216.917,A -85,B 0,C 180,E1 -20422.701,E2 -20422.701} C_VEL
LIN {X 0,Y 221.511,Z 216.889,A -85,B 0,C 180,E1 -20428.181,E2 -20428.181} C_VEL
LIN {X 0,Y 221.51,Z 216.89,A -85,B 0,C 180,E1 -20431.817,E2 -20431.817} C_VEL
LIN {X 0,Y 221.286,Z 216.917,A -85,B 0,C 180,E1 -20437.297,E2 -20437.297} C_VEL
LIN {X 0,Y 221.109,Z 216.944,A -85,B 0,C 180,E1 -20440.993,E2 -20440.993} C_VEL
LIN {X 0,Y 221.013,Z 216.953,A -85,B 0,C 180,E1 -20446.629,E2 -20446.629} C_VEL
LIN {X 0,Y 220.888,Z 216.97,A -85,B 0,C 180,E1 -20450.485,E2 -20450.485} C_VEL
LIN {X 0,Y 220.863,Z 216.972,A -85,B 0,C 180,E1 -20454.434,E2 -20454.434} C_VEL
LIN {X 0,Y 220.832,Z 216.978,A -85,B 0,C 180,E1 -20458.512,E2 -20458.512} C_VEL
LIN {X 0,Y 220.819,Z 216.976,A -85,B 0,C 180,E1 -20462.754,E2 -20462.754} C_VEL
LIN {X 0,Y 220.832,Z 216.975,A -85,B 0,C 180,E1 -20467.287,E2 -20467.287} C_VEL
LIN {X 0,Y 220.847,Z 216.971,A -85,B 0,C 180,E1 -20471.932,E2 -20471.932} C_VEL
LIN {X 0,Y 220.855,Z 216.972,A -85,B 0,C 180,E1 -20477.043,E2 -20477.043} C_VEL
LIN {X 0,Y 220.829,Z 216.976,A -85,B 0,C 180,E1 -20480.469,E2 -20480.469} C_VEL
LIN {X 0,Y 220.809,Z 216.978,A -85,B 0,C 180,E1 -20485.048,E2 -20485.048} C_VEL
LIN {X 0,Y 220.861,Z 216.969,A -85,B 0,C 180,E1 -20489.395,E2 -20489.395} C_VEL
LIN {X 0,Y 220.888,Z 216.969,A -85,B 0,C 180,E1 -20493.55,E2 -20493.55} C_VEL
LIN {X 0,Y 220.871,Z 216.968,A -85,B 0,C 180,E1 -20497.554,E2 -20497.554} C_VEL
LIN {X 0,Y 220.978,Z 216.957,A -85,B 0,C 180,E1 -20502.571,E2 -20502.571} C_VEL
LIN {X 0,Y 221.005,Z 216.953,A -85,B 0,C 180,E1 -20507.139,E2 -20507.139} C_VEL
LIN {X 0,Y 221.198,Z 216.929,A -85,B 0,C 180,E1 -20510.86,E2 -20510.86} C_VEL
LIN {X 0,Y 221.253,Z 216.921,A -85,B 0,C 180,E1 -20512.701,E2 -20512.701} C_VEL
LIN {X 0,Y 221.505,Z 216.892,A -85,B 0,C 180,E1 -20518.183,E2 -20518.183} C_VEL
LIN {X 0,Y 221.506,Z 216.891,A -85,B 0,C 180,E1 -20521.819,E2 -20521.819} C_VEL
LIN {X 0,Y 221.3,Z 216.919,A -85,B 0,C 180,E1 -20527.299,E2 -20527.299} C_VEL
LIN {X 0,Y 221.101,Z 216.939,A -85,B 0,C 180,E1 -20530.996,E2 -20530.996} C_VEL
LIN {X 0,Y 221.011,Z 216.953,A -85,B 0,C 180,E1 -20536.631,E2 -20536.631} C_VEL
LIN {X 0,Y 220.888,Z 216.967,A -85,B 0,C 180,E1 -20540.487,E2 -20540.487} C_VEL
LIN {X 0,Y 220.863,Z 216.971,A -85,B 0,C 180,E1 -20544.436,E2 -20544.436} C_VEL
LIN {X 0,Y 220.823,Z 216.975,A -85,B 0,C 180,E1 -20548.516,E2 -20548.516} C_VEL
LIN {X 0,Y 220.812,Z 216.978,A -85,B 0,C 180,E1 -20552.758,E2 -20552.758} C_VEL
LIN {X 0,Y 220.807,Z 216.981,A -85,B 0,C 180,E1 -20557.28,E2 -20557.28} C_VEL
LIN {X 0,Y 220.791,Z 216.981,A -85,B 0,C 180,E1 -20560.19,E2 -20560.19} C_VEL
LIN {X 0,Y 220.765,Z 216.985,A -85,B 0,C 180,E1 -20564.457,E2 -20564.457} C_VEL
LIN {X 0,Y 220.765,Z 216.985,A -85,B 0,C 180,E1 -20568.049,E2 -20568.049} C_VEL
LIN {X 0,Y 220.878,Z 217.159,A -85,B 0,C 180,E1 -20570.931,E2 -20570.931} C_VEL
LIN {X 0,Y 221.078,Z 218.064,A -85,B 0,C 180,E1 -20571.269,E2 -20571.269} C_VEL
LIN {X 0,Y 221.313,Z 221.751,A -85,B 0,C 180,E1 -20572.471,E2 -20572.471} C_VEL
LIN {X 0,Y 219.821,Z 228.218,A -85,B 0,C 180,E1 -20574.386,E2 -20574.386} C_VEL
LIN {X 0,Y 218.238,Z 234.75,A -85,B 0,C 180,E1 -20576.318,E2 -20576.318} C_VEL
LIN {X 0,Y 218.362,Z 238.55,A -85,B 0,C 180,E1 -20577.52,E2 -20577.52} C_VEL
LIN {X 0,Y 219.791,Z 245.306,A -85,B 0,C 180,E1 -20579.696,E2 -20579.696} C_VEL
LIN {X 0,Y 219.533,Z 248.902,A -85,B 0,C 180,E1 -20580.782,E2 -20580.782} C_VEL
LIN {X 0,Y 218.29,Z 255.276,A -85,B 0,C 180,E1 -20582.628,E2 -20582.628} C_VEL
LIN {X 0,Y 218.988,Z 275.563,A -85,B 0,C 180,E1 -20583.632,E2 -20583.632} C_VEL
LIN {X 0,Y 220.766,Z 302.659,A -85,B 0,C 180,E1 -20584.936,E2 -20584.936} C_VEL
LIN {X 0,Y 218.904,Z 357.585,A -85,B 0,C 180,E1 -20587.341,E2 -20587.341} C_VEL
LIN {X 0,Y 218.255,Z 369.004,A -85,B 0,C 180,E1 -20588.143,E2 -20588.143} C_VEL
LIN {X 0,Y 217.223,Z 381.576,A -85,B 0,C 180,E1 -20589.386,E2 -20589.386} C_VEL
LIN {X 0,Y 216.025,Z 393.706,A -85,B 0,C 180,E1 -20591.016,E2 -20591.016} C_VEL
LIN {X 0,Y 214.941,Z 404.506,A -85,B 0,C 180,E1 -20592.887,E2 -20592.887} C_VEL
LIN {X 0,Y 213.786,Z 415.188,A -85,B 0,C 180,E1 -20595.241,E2 -20595.241} C_VEL
LIN {X 0,Y 213.142,Z 423.811,A -85,B 0,C 180,E1 -20597.625,E2 -20597.625} C_VEL
LIN {X 0,Y 212.679,Z 432.062,A -85,B 0,C 180,E1 -20600.491,E2 -20600.491} C_VEL
LIN {X 0,Y 212.665,Z 438.194,A -85,B 0,C 180,E1 -20603.18,E2 -20603.18} C_VEL
LIN {X 0,Y 212.904,Z 443.492,A -85,B 0,C 180,E1 -20606.216,E2 -20606.216} C_VEL
LIN {X 0,Y 212.987,Z 446.025,A -85,B 0,C 180,E1 -20608.11,E2 -20608.11} C_VEL
LIN {X 0,Y 213.021,Z 447.982,A -85,B 0,C 180,E1 -20610.001,E2 -20610.001} C_VEL
LIN {X 0,Y 212.806,Z 449.389,A -85,B 0,C 180,E1 -20611.894,E2 -20611.894} C_VEL
LIN {X 0,Y 212.404,Z 450.325,A -85,B 0,C 180,E1 -20613.796,E2 -20613.796} C_VEL
LIN {X 0,Y 212.058,Z 450.857,A -85,B 0,C 180,E1 -20616.136,E2 -20616.136} C_VEL
LIN {X 0,Y 211.996,Z 450.546,A -85,B 0,C 180,E1 -20619.542,E2 -20619.542} C_VEL
LIN {X 0,Y 212.273,Z 449.83,A -85,B 0,C 180,E1 -20621.459,E2 -20621.459} C_VEL
LIN {X 0,Y 212.83,Z 448.695,A -85,B 0,C 180,E1 -20623.366,E2 -20623.366} C_VEL
LIN {X 0,Y 213.772,Z 447.163,A -85,B 0,C 180,E1 -20625.25,E2 -20625.25} C_VEL
LIN {X 0,Y 215.579,Z 444.076,A -85,B 0,C 180,E1 -20628.043,E2 -20628.043} C_VEL
LIN {X 0,Y 217.986,Z 439.983,A -85,B 0,C 180,E1 -20630.773,E2 -20630.773} C_VEL
LIN {X 0,Y 220.897,Z 434.827,A -85,B 0,C 180,E1 -20633.435,E2 -20633.435} C_VEL
LIN {X 0,Y 224.537,Z 428.406,A -85,B 0,C 180,E1 -20635.99,E2 -20635.99} C_VEL
LIN {X 0,Y 228.82,Z 420.443,A -85,B 0,C 180,E1 -20638.43,E2 -20638.43} C_VEL
LIN {X 0,Y 233.537,Z 410.705,A -85,B 0,C 180,E1 -20640.771,E2 -20640.771} C_VEL
LIN {X 0,Y 237.932,Z 400.656,A -85,B 0,C 180,E1 -20642.621,E2 -20642.621} C_VEL
LIN {X 0,Y 242.302,Z 389.436,A -85,B 0,C 180,E1 -20644.193,E2 -20644.193} C_VEL
LIN {X 0,Y 245.884,Z 378.508,A -85,B 0,C 180,E1 -20645.367,E2 -20645.367} C_VEL
LIN {X 0,Y 249.391,Z 365.523,A -85,B 0,C 180,E1 -20646.411,E2 -20646.411} C_VEL
LIN {X 0,Y 252.031,Z 351.822,A -85,B 0,C 180,E1 -20647.213,E2 -20647.213} C_VEL
LIN {X 0,Y 256.913,Z 311.458,A -85,B 0,C 180,E1 -20648.853,E2 -20648.853} C_VEL
LIN {X 0,Y 256.974,Z 299.765,A -85,B 0,C 180,E1 -20649.833,E2 -20649.833} C_VEL
LIN {X 0,Y 256.822,Z 293.596,A -85,B 0,C 180,E1 -20650.47,E2 -20650.47} C_VEL
LIN {X 0,Y 254.427,Z 287.39,A -85,B 0,C 180,E1 -20652.113,E2 -20652.113} C_VEL
LIN {X 0,Y 252.388,Z 282.755,A -85,B 0,C 180,E1 -20653.669,E2 -20653.669} C_VEL
LIN {X 0,Y 250.57,Z 279.187,A -85,B 0,C 180,E1 -20655.13,E2 -20655.13} C_VEL
LIN {X 0,Y 248.269,Z 274.33,A -85,B 0,C 180,E1 -20657.476,E2 -20657.476} C_VEL
LIN {X 0,Y 245.579,Z 269.589,A -85,B 0,C 180,E1 -20661.107,E2 -20661.107} C_VEL
LIN {X 0,Y 244.429,Z 267.035,A -85,B 0,C 180,E1 -20664.137,E2 -20664.137} C_VEL
LIN {X 0,Y 244.061,Z 266.313,A -85,B 0,C 180,E1 -20666.829,E2 -20666.829} C_VEL
LIN {X 0,Y 244.486,Z 266.456,A -85,B 0,C 180,E1 -20669.586,E2 -20669.586} C_VEL
LIN {X 0,Y 246.077,Z 268.341,A -85,B 0,C 180,E1 -20673.099,E2 -20673.099} C_VEL
LIN {X 0,Y 247.7,Z 270.497,A -85,B 0,C 180,E1 -20675.302,E2 -20675.302} C_VEL
LIN {X 0,Y 250.644,Z 274.979,A -85,B 0,C 180,E1 -20678.302,E2 -20678.302} C_VEL
LIN {X 0,Y 253.255,Z 279.415,A -85,B 0,C 180,E1 -20680.405,E2 -20680.405} C_VEL
LIN {X 0,Y 255.727,Z 284.186,A -85,B 0,C 180,E1 -20682.181,E2 -20682.181} C_VEL
LIN {X 0,Y 258.603,Z 290.424,A -85,B 0,C 180,E1 -20684.056,E2 -20684.056} C_VEL
LIN {X 0,Y 253.044,Z 333.064,A -85,B 0,C 180,E1 -20686.031,E2 -20686.031} C_VEL
LIN {X 0,Y 250.791,Z 345.832,A -85,B 0,C 180,E1 -20686.931,E2 -20686.931} C_VEL
LIN {X 0,Y 247.825,Z 358.08,A -85,B 0,C 180,E1 -20688.135,E2 -20688.135} C_VEL
LIN {X 0,Y 244.813,Z 367.913,A -85,B 0,C 180,E1 -20689.389,E2 -20689.389} C_VEL
LIN {X 0,Y 241.077,Z 378.235,A -85,B 0,C 180,E1 -20691.067,E2 -20691.067} C_VEL
LIN {X 0,Y 237.576,Z 386.456,A -85,B 0,C 180,E1 -20692.777,E2 -20692.777} C_VEL
LIN {X 0,Y 233.691,Z 394.253,A -85,B 0,C 180,E1 -20694.823,E2 -20694.823} C_VEL
LIN {X 0,Y 230.142,Z 400.515,A -85,B 0,C 180,E1 -20696.936,E2 -20696.936} C_VEL
LIN {X 0,Y 226.876,Z 405.566,A -85,B 0,C 180,E1 -20699.112,E2 -20699.112} C_VEL
LIN {X 0,Y 223.355,Z 410.197,A -85,B 0,C 180,E1 -20701.802,E2 -20701.802} C_VEL
LIN {X 0,Y 221.301,Z 412.486,A -85,B 0,C 180,E1 -20703.641,E2 -20703.641} C_VEL
LIN {X 0,Y 219.045,Z 414.515,A -85,B 0,C 180,E1 -20705.936,E2 -20705.936} C_VEL
LIN {X 0,Y 216.408,Z 416.01,A -85,B 0,C 180,E1 -20709.344,E2 -20709.344} C_VEL
LIN {X 0,Y 215.119,Z 416.058,A -85,B 0,C 180,E1 -20711.443,E2 -20711.443} C_VEL
LIN {X 0,Y 214.202,Z 415.627,A -85,B 0,C 180,E1 -20713.277,E2 -20713.277} C_VEL
LIN {X 0,Y 212.92,Z 413.451,A -85,B 0,C 180,E1 -20716.817,E2 -20716.817} C_VEL
LIN {X 0,Y 212.437,Z 410.845,A -85,B 0,C 180,E1 -20719.318,E2 -20719.318} C_VEL
LIN {X 0,Y 212.296,Z 405.945,A -85,B 0,C 180,E1 -20722.612,E2 -20722.612} C_VEL
LIN {X 0,Y 212.538,Z 400.231,A -85,B 0,C 180,E1 -20725.458,E2 -20725.458} C_VEL
LIN {X 0,Y 213.001,Z 393.567,A -85,B 0,C 180,E1 -20728.045,E2 -20728.045} C_VEL
LIN {X 0,Y 213.678,Z 385.184,A -85,B 0,C 180,E1 -20730.642,E2 -20730.642} C_VEL
LIN {X 0,Y 214.553,Z 375.589,A -85,B 0,C 180,E1 -20732.994,E2 -20732.994} C_VEL
LIN {X 0,Y 215.559,Z 364.443,A -85,B 0,C 180,E1 -20735.134,E2 -20735.134} C_VEL
LIN {X 0,Y 216.533,Z 352.548,A -85,B 0,C 180,E1 -20736.901,E2 -20736.901} C_VEL
LIN {X 0,Y 217.4,Z 340.286,A -85,B 0,C 180,E1 -20738.275,E2 -20738.275} C_VEL
LIN {X 0,Y 218.044,Z 327.677,A -85,B 0,C 180,E1 -20739.292,E2 -20739.292} C_VEL
LIN {X 0,Y 218.853,Z 302.777,A -85,B 0,C 180,E1 -20740.562,E2 -20740.562} C_VEL
LIN {X 0,Y 220.456,Z 263.292,A -85,B 0,C 180,E1 -20742.431,E2 -20742.431} C_VEL
LIN {X 0,Y 217.316,Z 236.252,A -85,B 0,C 180,E1 -20743.98,E2 -20743.98} C_VEL
LIN {X 0,Y 216.288,Z 229.961,A -85,B 0,C 180,E1 -20746.219,E2 -20746.219} C_VEL
LIN {X 0,Y 213.849,Z 218.029,A -85,B 0,C 180,E1 -20750.905,E2 -20750.905} C_VEL
LIN {X 0,Y 213.76,Z 217.859,A -85,B 0,C 180,E1 -20756.017,E2 -20756.017} C_VEL
LIN {X 0,Y 213.78,Z 217.854,A -85,B 0,C 180,E1 -20760.453,E2 -20760.453} C_VEL
LIN {X 0,Y 213.801,Z 217.851,A -85,B 0,C 180,E1 -20764.7,E2 -20764.7} C_VEL
LIN {X 0,Y 213.812,Z 217.85,A -85,B 0,C 180,E1 -20768.802,E2 -20768.802} C_VEL
LIN {X 0,Y 213.943,Z 217.833,A -85,B 0,C 180,E1 -20772.802,E2 -20772.802} C_VEL
LIN {X 0,Y 213.979,Z 217.83,A -85,B 0,C 180,E1 -20776.707,E2 -20776.707} C_VEL
LIN {X 0,Y 214.195,Z 217.8,A -85,B 0,C 180,E1 -20780.556,E2 -20780.556} C_VEL
LIN {X 0,Y 214.11,Z 217.813,A -85,B 0,C 180,E1 -20784.347,E2 -20784.347} C_VEL
LIN {X 0,Y 214.444,Z 217.77,A -85,B 0,C 180,E1 -20788.121,E2 -20788.121} C_VEL
LIN {X 0,Y 214.548,Z 217.755,A -85,B 0,C 180,E1 -20789.999,E2 -20789.999} C_VEL
LIN {X 0,Y 214.444,Z 217.771,A -85,B 0,C 180,E1 -20791.877,E2 -20791.877} C_VEL
LIN {X 0,Y 214.224,Z 217.796,A -85,B 0,C 180,E1 -20797.539,E2 -20797.539} C_VEL
LIN {X 0,Y 214.041,Z 217.822,A -85,B 0,C 180,E1 -20801.361,E2 -20801.361} C_VEL
LIN {X 0,Y 213.93,Z 217.834,A -85,B 0,C 180,E1 -20805.236,E2 -20805.236} C_VEL
LIN {X 0,Y 213.836,Z 217.848,A -85,B 0,C 180,E1 -20809.186,E2 -20809.186} C_VEL
LIN {X 0,Y 213.843,Z 217.845,A -85,B 0,C 180,E1 -20813.226,E2 -20813.226} C_VEL
LIN {X 0,Y 213.824,Z 217.848,A -85,B 0,C 180,E1 -20817.449,E2 -20817.449} C_VEL
LIN {X 0,Y 213.774,Z 217.853,A -85,B 0,C 180,E1 -20821.735,E2 -20821.735} C_VEL
LIN {X 0,Y 213.749,Z 217.859,A -85,B 0,C 180,E1 -20826.285,E2 -20826.285} C_VEL
LIN {X 0,Y 213.788,Z 217.85,A -85,B 0,C 180,E1 -20831.105,E2 -20831.105} C_VEL
LIN {X 0,Y 213.802,Z 217.85,A -85,B 0,C 180,E1 -20833.684,E2 -20833.684} C_VEL
LIN {X 0,Y 213.805,Z 217.854,A -85,B 0,C 180,E1 -20836.348,E2 -20836.348} C_VEL
LIN {X 0,Y 213.764,Z 217.854,A -85,B 0,C 180,E1 -20841.343,E2 -20841.343} C_VEL
LIN {X 0,Y 213.763,Z 217.858,A -85,B 0,C 180,E1 -20846.02,E2 -20846.02} C_VEL
LIN {X 0,Y 213.774,Z 217.856,A -85,B 0,C 180,E1 -20850.454,E2 -20850.454} C_VEL
LIN {X 0,Y 213.794,Z 217.851,A -85,B 0,C 180,E1 -20854.702,E2 -20854.702} C_VEL
LIN {X 0,Y 213.806,Z 217.85,A -85,B 0,C 180,E1 -20858.804,E2 -20858.804} C_VEL
LIN {X 0,Y 213.937,Z 217.834,A -85,B 0,C 180,E1 -20862.804,E2 -20862.804} C_VEL
LIN {X 0,Y 213.946,Z 217.832,A -85,B 0,C 180,E1 -20866.707,E2 -20866.707} C_VEL
LIN {X 0,Y 214.135,Z 217.809,A -85,B 0,C 180,E1 -20870.556,E2 -20870.556} C_VEL
LIN {X 0,Y 214.094,Z 217.813,A -85,B 0,C 180,E1 -20874.349,E2 -20874.349} C_VEL
LIN {X 0,Y 214.439,Z 217.773,A -85,B 0,C 180,E1 -20878.123,E2 -20878.123} C_VEL
LIN {X 0,Y 214.544,Z 217.759,A -85,B 0,C 180,E1 -20880.001,E2 -20880.001} C_VEL
LIN {X 0,Y 214.439,Z 217.771,A -85,B 0,C 180,E1 -20881.879,E2 -20881.879} C_VEL
LIN {X 0,Y 214.235,Z 217.8,A -85,B 0,C 180,E1 -20887.541,E2 -20887.541} C_VEL
LIN {X 0,Y 214.018,Z 217.823,A -85,B 0,C 180,E1 -20891.364,E2 -20891.364} C_VEL
LIN {X 0,Y 213.929,Z 217.838,A -85,B 0,C 180,E1 -20895.238,E2 -20895.238} C_VEL
LIN {X 0,Y 213.835,Z 217.846,A -85,B 0,C 180,E1 -20899.189,E2 -20899.189} C_VEL
LIN {X 0,Y 213.843,Z 217.849,A -85,B 0,C 180,E1 -20903.228,E2 -20903.228} C_VEL
LIN {X 0,Y 213.825,Z 217.849,A -85,B 0,C 180,E1 -20907.451,E2 -20907.451} C_VEL
LIN {X 0,Y 213.764,Z 217.856,A -85,B 0,C 180,E1 -20911.739,E2 -20911.739} C_VEL
LIN {X 0,Y 213.74,Z 217.858,A -85,B 0,C 180,E1 -20916.29,E2 -20916.29} C_VEL
LIN {X 0,Y 213.708,Z 217.866,A -85,B 0,C 180,E1 -20921.127,E2 -20921.127} C_VEL
LIN {X 0,Y 213.701,Z 217.865,A -85,B 0,C 180,E1 -20923.681,E2 -20923.681} C_VEL
LIN {X 0,Y 213.701,Z 217.866,A -85,B 0,C 180,E1 -20926.347,E2 -20926.347} C_VEL
LIN {X 0,Y 213.79,Z 218.059,A -85,B 0,C 180,E1 -20930.482,E2 -20930.482} C_VEL
LIN {X 0,Y 216.275,Z 228.998,A -85,B 0,C 180,E1 -20934.332,E2 -20934.332} C_VEL
LIN {X 0,Y 218.362,Z 238.55,A -85,B 0,C 180,E1 -20937.52,E2 -20937.52} C_VEL
LIN {X 0,Y 218.163,Z 241.094,A -85,B 0,C 180,E1 -20938.298,E2 -20938.298} C_VEL
LIN {X 0,Y 216.408,Z 244.533,A -85,B 0,C 180,E1 -20939.258,E2 -20939.258} C_VEL
LIN {X 0,Y 212.454,Z 250.601,A -85,B 0,C 180,E1 -20940.936,E2 -20940.936} C_VEL
LIN {X 0,Y 211.843,Z 252.389,A -85,B 0,C 180,E1 -20941.469,E2 -20941.469} C_VEL
LIN {X 0,Y 211.336,Z 255.346,A -85,B 0,C 180,E1 -20942.255,E2 -20942.255} C_VEL
LIN {X 0,Y 212.036,Z 276.411,A -85,B 0,C 180,E1 -20943.318,E2 -20943.318} C_VEL
LIN {X 0,Y 213.765,Z 303.423,A -85,B 0,C 180,E1 -20944.664,E2 -20944.664} C_VEL
LIN {X 0,Y 211.858,Z 357.409,A -85,B 0,C 180,E1 -20947.125,E2 -20947.125} C_VEL
LIN {X 0,Y 211.144,Z 369.383,A -85,B 0,C 180,E1 -20948.011,E2 -20948.011} C_VEL
LIN {X 0,Y 210.193,Z 381.037,A -85,B 0,C 180,E1 -20949.219,E2 -20949.219} C_VEL
LIN {X 0,Y 208.984,Z 392.884,A -85,B 0,C 180,E1 -20950.861,E2 -20950.861} C_VEL
LIN {X 0,Y 207.882,Z 403.734,A -85,B 0,C 180,E1 -20952.795,E2 -20952.795} C_VEL
LIN {X 0,Y 206.729,Z 414.406,A -85,B 0,C 180,E1 -20955.23,E2 -20955.23} C_VEL
LIN {X 0,Y 206.105,Z 423.043,A -85,B 0,C 180,E1 -20957.696,E2 -20957.696} C_VEL
LIN {X 0,Y 205.705,Z 430.038,A -85,B 0,C 180,E1 -20960.166,E2 -20960.166} C_VEL
LIN {X 0,Y 205.674,Z 436.582,A -85,B 0,C 180,E1 -20963.031,E2 -20963.031} C_VEL
LIN {X 0,Y 205.884,Z 441.996,A -85,B 0,C 180,E1 -20966.087,E2 -20966.087} C_VEL
LIN {X 0,Y 205.975,Z 445.767,A -85,B 0,C 180,E1 -20969.024,E2 -20969.024} C_VEL
LIN {X 0,Y 206.014,Z 446.751,A -85,B 0,C 180,E1 -20970.001,E2 -20970.001} C_VEL
LIN {X 0,Y 205.772,Z 448.287,A -85,B 0,C 180,E1 -20971.959,E2 -20971.959} C_VEL
LIN {X 0,Y 205.348,Z 449.308,A -85,B 0,C 180,E1 -20973.926,E2 -20973.926} C_VEL
LIN {X 0,Y 205.012,Z 449.982,A -85,B 0,C 180,E1 -20976.193,E2 -20976.193} C_VEL
LIN {X 0,Y 204.965,Z 449.873,A -85,B 0,C 180,E1 -20979.873,E2 -20979.873} C_VEL
LIN {X 0,Y 205.887,Z 448.254,A -85,B 0,C 180,E1 -20983.826,E2 -20983.826} C_VEL
LIN {X 0,Y 206.894,Z 446.863,A -85,B 0,C 180,E1 -20985.77,E2 -20985.77} C_VEL
LIN {X 0,Y 208.827,Z 443.996,A -85,B 0,C 180,E1 -20988.647,E2 -20988.647} C_VEL
LIN {X 0,Y 211.348,Z 440.149,A -85,B 0,C 180,E1 -20991.457,E2 -20991.457} C_VEL
LIN {X 0,Y 214.42,Z 435.22,A -85,B 0,C 180,E1 -20994.188,E2 -20994.188} C_VEL
LIN {X 0,Y 218.962,Z 427.922,A -85,B 0,C 180,E1 -20997.219,E2 -20997.219} C_VEL
LIN {X 0,Y 223.465,Z 420.153,A -85,B 0,C 180,E1 -20999.693,E2 -20999.693} C_VEL
LIN {X 0,Y 228.458,Z 410.496,A -85,B 0,C 180,E1 -21002.051,E2 -21002.051} C_VEL
LIN {X 0,Y 233.095,Z 400.574,A -85,B 0,C 180,E1 -21003.904,E2 -21003.904} C_VEL
LIN {X 0,Y 237.108,Z 390.978,A -85,B 0,C 180,E1 -21005.31,E2 -21005.31} C_VEL
LIN {X 0,Y 241.381,Z 379.12,A -85,B 0,C 180,E1 -21006.647,E2 -21006.647} C_VEL
LIN {X 0,Y 244.733,Z 367.677,A -85,B 0,C 180,E1 -21007.608,E2 -21007.608} C_VEL
LIN {X 0,Y 247.66,Z 354.474,A -85,B 0,C 180,E1 -21008.438,E2 -21008.438} C_VEL
LIN {X 0,Y 250.392,Z 334.817,A -85,B 0,C 180,E1 -21009.275,E2 -21009.275} C_VEL
LIN {X 0,Y 253.193,Z 312.429,A -85,B 0,C 180,E1 -21010.206,E2 -21010.206} C_VEL
LIN {X 0,Y 253.402,Z 301.38,A -85,B 0,C 180,E1 -21011.176,E2 -21011.176} C_VEL
LIN {X 0,Y 253.31,Z 297.602,A -85,B 0,C 180,E1 -21011.591,E2 -21011.591} C_VEL
LIN {X 0,Y 250.989,Z 291.165,A -85,B 0,C 180,E1 -21013.432,E2 -21013.432} C_VEL
LIN {X 0,Y 248.562,Z 285.851,A -85,B 0,C 180,E1 -21015.498,E2 -21015.498} C_VEL
LIN {X 0,Y 246.208,Z 280.769,A -85,B 0,C 180,E1 -21017.999,E2 -21017.999} C_VEL
LIN {X 0,Y 243.886,Z 276.205,A -85,B 0,C 180,E1 -21021.549,E2 -21021.549} C_VEL
LIN {X 0,Y 242.914,Z 273.901,A -85,B 0,C 180,E1 -21024.39,E2 -21024.39} C_VEL
LIN {X 0,Y 242.612,Z 273.254,A -85,B 0,C 180,E1 -21027.149,E2 -21027.149} C_VEL
LIN {X 0,Y 243.159,Z 273.597,A -85,B 0,C 180,E1 -21030.123,E2 -21030.123} C_VEL
LIN {X 0,Y 244.754,Z 275.651,A -85,B 0,C 180,E1 -21033.422,E2 -21033.422} C_VEL
LIN {X 0,Y 245.931,Z 277.344,A -85,B 0,C 180,E1 -21035.056,E2 -21035.056} C_VEL
LIN {X 0,Y 248.56,Z 281.548,A -85,B 0,C 180,E1 -21037.893,E2 -21037.893} C_VEL
LIN {X 0,Y 250.745,Z 285.509,A -85,B 0,C 180,E1 -21039.809,E2 -21039.809} C_VEL
LIN {X 0,Y 253.454,Z 291.074,A -85,B 0,C 180,E1 -21041.905,E2 -21041.905} C_VEL
LIN {X 0,Y 254.766,Z 294.08,A -85,B 0,C 180,E1 -21042.814,E2 -21042.814} C_VEL
LIN {X 0,Y 249.203,Z 333.939,A -85,B 0,C 180,E1 -21044.682,E2 -21044.682} C_VEL
LIN {X 0,Y 246.643,Z 347.356,A -85,B 0,C 180,E1 -21045.656,E2 -21045.656} C_VEL
LIN {X 0,Y 243.521,Z 359.483,A -85,B 0,C 180,E1 -21046.863,E2 -21046.863} C_VEL
LIN {X 0,Y 240.192,Z 369.618,A -85,B 0,C 180,E1 -21048.18,E2 -21048.18} C_VEL
LIN {X 0,Y 236.582,Z 378.922,A -85,B 0,C 180,E1 -21049.732,E2 -21049.732} C_VEL
LIN {X 0,Y 233.092,Z 386.589,A -85,B 0,C 180,E1 -21051.328,E2 -21051.328} C_VEL
LIN {X 0,Y 228.943,Z 394.509,A -85,B 0,C 180,E1 -21053.389,E2 -21053.389} C_VEL
LIN {X 0,Y 225.041,Z 400.998,A -85,B 0,C 180,E1 -21055.551,E2 -21055.551} C_VEL
LIN {X 0,Y 220.913,Z 406.872,A -85,B 0,C 180,E1 -21058.176,E2 -21058.176} C_VEL
LIN {X 0,Y 217.875,Z 410.562,A -85,B 0,C 180,E1 -21060.369,E2 -21060.369} C_VEL
LIN {X 0,Y 216.042,Z 412.536,A -85,B 0,C 180,E1 -21061.863,E2 -21061.863} C_VEL
LIN {X 0,Y 213.946,Z 414.457,A -85,B 0,C 180,E1 -21063.766,E2 -21063.766} C_VEL
LIN {X 0,Y 211.946,Z 415.905,A -85,B 0,C 180,E1 -21065.848,E2 -21065.848} C_VEL
LIN {X 0,Y 210.446,Z 416.613,A -85,B 0,C 180,E1 -21067.676,E2 -21067.676} C_VEL
LIN {X 0,Y 209.028,Z 416.907,A -85,B 0,C 180,E1 -21069.677,E2 -21069.677} C_VEL
LIN {X 0,Y 207.847,Z 416.629,A -85,B 0,C 180,E1 -21071.704,E2 -21071.704} C_VEL
LIN {X 0,Y 206.851,Z 415.842,A -85,B 0,C 180,E1 -21073.758,E2 -21073.758} C_VEL
LIN {X 0,Y 205.766,Z 413.453,A -85,B 0,C 180,E1 -21076.989,E2 -21076.989} C_VEL
LIN {X 0,Y 205.262,Z 409.984,A -85,B 0,C 180,E1 -21080.022,E2 -21080.022} C_VEL
LIN {X 0,Y 205.24,Z 404.865,A -85,B 0,C 180,E1 -21083.202,E2 -21083.202} C_VEL
LIN {X 0,Y 205.531,Z 399.307,A -85,B 0,C 180,E1 -21085.846,E2 -21085.846} C_VEL
LIN {X 0,Y 206.016,Z 392.23,A -85,B 0,C 180,E1 -21088.527,E2 -21088.527} C_VEL
LIN {X 0,Y 206.725,Z 383.798,A -85,B 0,C 180,E1 -21091.077,E2 -21091.077} C_VEL
LIN {X 0,Y 207.607,Z 374.302,A -85,B 0,C 180,E1 -21093.373,E2 -21093.373} C_VEL
LIN {X 0,Y 208.548,Z 363.9,A -85,B 0,C 180,E1 -21095.386,E2 -21095.386} C_VEL
LIN {X 0,Y 209.499,Z 352.281,A -85,B 0,C 180,E1 -21097.144,E2 -21097.144} C_VEL
LIN {X 0,Y 210.414,Z 339.24,A -85,B 0,C 180,E1 -21098.621,E2 -21098.621} C_VEL
LIN {X 0,Y 211.1,Z 325.499,A -85,B 0,C 180,E1 -21099.693,E2 -21099.693} C_VEL
LIN {X 0,Y 213.406,Z 263.222,A -85,B 0,C 180,E1 -21102.8,E2 -21102.8} C_VEL
LIN {X 0,Y 210.279,Z 236.574,A -85,B 0,C 180,E1 -21104.384,E2 -21104.384} C_VEL
LIN {X 0,Y 208.359,Z 226.547,A -85,B 0,C 180,E1 -21108.167,E2 -21108.167} C_VEL
LIN {X 0,Y 206.858,Z 219.14,A -85,B 0,C 180,E1 -21111.159,E2 -21111.159} C_VEL
LIN {X 0,Y 206.748,Z 218.733,A -85,B 0,C 180,E1 -21111.84,E2 -21111.84} C_VEL
LIN {X 0,Y 206.704,Z 218.737,A -85,B 0,C 180,E1 -21117.042,E2 -21117.042} C_VEL
LIN {X 0,Y 206.766,Z 218.729,A -85,B 0,C 180,E1 -21122.095,E2 -21122.095} C_VEL
LIN {X 0,Y 206.785,Z 218.726,A -85,B 0,C 180,E1 -21126.582,E2 -21126.582} C_VEL
LIN {X 0,Y 206.872,Z 218.713,A -85,B 0,C 180,E1 -21132.195,E2 -21132.195} C_VEL
LIN {X 0,Y 206.913,Z 218.709,A -85,B 0,C 180,E1 -21136.244,E2 -21136.244} C_VEL
LIN {X 0,Y 207.131,Z 218.68,A -85,B 0,C 180,E1 -21140.231,E2 -21140.231} C_VEL
LIN {X 0,Y 207.073,Z 218.689,A -85,B 0,C 180,E1 -21144.155,E2 -21144.155} C_VEL
LIN {X 0,Y 207.381,Z 218.649,A -85,B 0,C 180,E1 -21148.057,E2 -21148.057} C_VEL
LIN {X 0,Y 207.513,Z 218.631,A -85,B 0,C 180,E1 -21149.999,E2 -21149.999} C_VEL
LIN {X 0,Y 207.38,Z 218.65,A -85,B 0,C 180,E1 -21151.941,E2 -21151.941} C_VEL
LIN {X 0,Y 207.164,Z 218.674,A -85,B 0,C 180,E1 -21157.798,E2 -21157.798} C_VEL
LIN {X 0,Y 206.978,Z 218.701,A -85,B 0,C 180,E1 -21161.754,E2 -21161.754} C_VEL
LIN {X 0,Y 206.863,Z 218.713,A -85,B 0,C 180,E1 -21165.769,E2 -21165.769} C_VEL
LIN {X 0,Y 206.78,Z 218.726,A -85,B 0,C 180,E1 -21169.868,E2 -21169.868} C_VEL
LIN {X 0,Y 206.759,Z 218.727,A -85,B 0,C 180,E1 -21174.071,E2 -21174.071} C_VEL
LIN {X 0,Y 206.739,Z 218.733,A -85,B 0,C 180,E1 -21178.418,E2 -21178.418} C_VEL
LIN {X 0,Y 206.704,Z 218.733,A -85,B 0,C 180,E1 -21182.955,E2 -21182.955} C_VEL
LIN {X 0,Y 206.719,Z 218.734,A -85,B 0,C 180,E1 -21187.729,E2 -21187.729} C_VEL
LIN {X 0,Y 206.717,Z 218.73,A -85,B 0,C 180,E1 -21191.588,E2 -21191.588} C_VEL
LIN {X 0,Y 206.711,Z 218.734,A -85,B 0,C 180,E1 -21195.557,E2 -21195.557} C_VEL
LIN {X 0,Y 206.697,Z 218.734,A -85,B 0,C 180,E1 -21199.759,E2 -21199.759} C_VEL
LIN {X 0,Y 206.715,Z 218.736,A -85,B 0,C 180,E1 -21202.269,E2 -21202.269} C_VEL
LIN {X 0,Y 206.703,Z 218.734,A -85,B 0,C 180,E1 -21207.044,E2 -21207.044} C_VEL
LIN {X 0,Y 206.76,Z 218.732,A -85,B 0,C 180,E1 -21212.096,E2 -21212.096} C_VEL
LIN {X 0,Y 206.779,Z 218.723,A -85,B 0,C 180,E1 -21216.584,E2 -21216.584} C_VEL
LIN {X 0,Y 206.867,Z 218.716,A -85,B 0,C 180,E1 -21222.197,E2 -21222.197} C_VEL
LIN {X 0,Y 206.889,Z 218.712,A -85,B 0,C 180,E1 -21226.245,E2 -21226.245} C_VEL
LIN {X 0,Y 207.093,Z 218.688,A -85,B 0,C 180,E1 -21230.232,E2 -21230.232} C_VEL
LIN {X 0,Y 207.055,Z 218.691,A -85,B 0,C 180,E1 -21234.157,E2 -21234.157} C_VEL
LIN {X 0,Y 207.375,Z 218.653,A -85,B 0,C 180,E1 -21238.059,E2 -21238.059} C_VEL
LIN {X 0,Y 207.509,Z 218.635,A -85,B 0,C 180,E1 -21240.001,E2 -21240.001} C_VEL
LIN {X 0,Y 207.376,Z 218.65,A -85,B 0,C 180,E1 -21241.943,E2 -21241.943} C_VEL
LIN {X 0,Y 207.173,Z 218.678,A -85,B 0,C 180,E1 -21247.8,E2 -21247.8} C_VEL
LIN {X 0,Y 206.938,Z 218.707,A -85,B 0,C 180,E1 -21251.758,E2 -21251.758} C_VEL
LIN {X 0,Y 206.862,Z 218.717,A -85,B 0,C 180,E1 -21255.772,E2 -21255.772} C_VEL
LIN {X 0,Y 206.779,Z 218.725,A -85,B 0,C 180,E1 -21259.87,E2 -21259.87} C_VEL
LIN {X 0,Y 206.759,Z 218.728,A -85,B 0,C 180,E1 -21264.074,E2 -21264.074} C_VEL
LIN {X 0,Y 206.733,Z 218.73,A -85,B 0,C 180,E1 -21268.421,E2 -21268.421} C_VEL
LIN {X 0,Y 206.695,Z 218.738,A -85,B 0,C 180,E1 -21272.959,E2 -21272.959} C_VEL
LIN {X 0,Y 206.676,Z 218.74,A -85,B 0,C 180,E1 -21277.742,E2 -21277.742} C_VEL
LIN {X 0,Y 206.638,Z 218.745,A -85,B 0,C 180,E1 -21281.564,E2 -21281.564} C_VEL
LIN {X 0,Y 206.629,Z 218.747,A -85,B 0,C 180,E1 -21285.584,E2 -21285.584} C_VEL
LIN {X 0,Y 206.748,Z 218.952,A -85,B 0,C 180,E1 -21290.035,E2 -21290.035} C_VEL
LIN {X 0,Y 209.33,Z 230.33,A -85,B 0,C 180,E1 -21294.161,E2 -21294.161} C_VEL
LIN {X 0,Y 212.228,Z 243.696,A -85,B 0,C 180,E1 -21298.732,E2 -21298.732} C_VEL
LIN {X 0,Y 212.789,Z 246.978,A -85,B 0,C 180,E1 -21299.81,E2 -21299.81} C_VEL
LIN {X 0,Y 211.843,Z 252.389,A -85,B 0,C 180,E1 -21301.469,E2 -21301.469} C_VEL
LIN {X 0,Y 211.01,Z 254.913,A -85,B 0,C 180,E1 -21301.989,E2 -21301.989} C_VEL
LIN {X 0,Y 209.223,Z 258.9,A -85,B 0,C 180,E1 -21302.329,E2 -21302.329} C_VEL
LIN {X 0,Y 206.082,Z 267.125,A -85,B 0,C 180,E1 -21302.535,E2 -21302.535} C_VEL
LIN {X 0,Y 205.268,Z 274.233,A -85,B 0,C 180,E1 -21302.825,E2 -21302.825} C_VEL
LIN {X 0,Y 205.438,Z 282.429,A -85,B 0,C 180,E1 -21303.258,E2 -21303.258} C_VEL
LIN {X 0,Y 206.779,Z 303.048,A -85,B 0,C 180,E1 -21304.322,E2 -21304.322} C_VEL
LIN {X 0,Y 204.819,Z 356.831,A -85,B 0,C 180,E1 -21306.894,E2 -21306.894} C_VEL
LIN {X 0,Y 204.17,Z 368.074,A -85,B 0,C 180,E1 -21307.752,E2 -21307.752} C_VEL
LIN {X 0,Y 203.095,Z 380.825,A -85,B 0,C 180,E1 -21309.121,E2 -21309.121} C_VEL
LIN {X 0,Y 201.838,Z 393.341,A -85,B 0,C 180,E1 -21310.949,E2 -21310.949} C_VEL
LIN {X 0,Y 200.731,Z 403.888,A -85,B 0,C 180,E1 -21312.95,E2 -21312.95} C_VEL
LIN {X 0,Y 199.692,Z 413.45,A -85,B 0,C 180,E1 -21315.219,E2 -21315.219} C_VEL
LIN {X 0,Y 199.078,Z 422.161,A -85,B 0,C 180,E1 -21317.773,E2 -21317.773} C_VEL
LIN {X 0,Y 198.691,Z 429.191,A -85,B 0,C 180,E1 -21320.329,E2 -21320.329} C_VEL
LIN {X 0,Y 198.681,Z 435.924,A -85,B 0,C 180,E1 -21323.377,E2 -21323.377} C_VEL
LIN {X 0,Y 198.867,Z 440.406,A -85,B 0,C 180,E1 -21325.948,E2 -21325.948} C_VEL
LIN {X 0,Y 199.006,Z 444.427,A -85,B 0,C 180,E1 -21328.99,E2 -21328.99} C_VEL
LIN {X 0,Y 199.015,Z 445.468,A -85,B 0,C 180,E1 -21330.001,E2 -21330.001} C_VEL
LIN {X 0,Y 198.746,Z 447.126,A -85,B 0,C 180,E1 -21332.028,E2 -21332.028} C_VEL
LIN {X 0,Y 198.311,Z 448.271,A -85,B 0,C 180,E1 -21334.066,E2 -21334.066} C_VEL
LIN {X 0,Y 197.97,Z 448.991,A -85,B 0,C 180,E1 -21336.266,E2 -21336.266} C_VEL
LIN {X 0,Y 197.953,Z 449.168,A -85,B 0,C 180,E1 -21340.226,E2 -21340.226} C_VEL
LIN {X 0,Y 198.309,Z 448.676,A -85,B 0,C 180,E1 -21342.278,E2 -21342.278} C_VEL
LIN {X 0,Y 198.965,Z 447.779,A -85,B 0,C 180,E1 -21344.317,E2 -21344.317} C_VEL
LIN {X 0,Y 201.299,Z 444.864,A -85,B 0,C 180,E1 -21348.315,E2 -21348.315} C_VEL
LIN {X 0,Y 204.319,Z 440.832,A -85,B 0,C 180,E1 -21351.761,E2 -21351.761} C_VEL
LIN {X 0,Y 207.973,Z 435.584,A -85,B 0,C 180,E1 -21354.988,E2 -21354.988} C_VEL
LIN {X 0,Y 211.962,Z 429.787,A -85,B 0,C 180,E1 -21357.659,E2 -21357.659} C_VEL
LIN {X 0,Y 216.585,Z 422.61,A -85,B 0,C 180,E1 -21360.197,E2 -21360.197} C_VEL
LIN {X 0,Y 221.683,Z 413.774,A -85,B 0,C 180,E1 -21362.613,E2 -21362.613} C_VEL
LIN {X 0,Y 226.854,Z 403.878,A -85,B 0,C 180,E1 -21364.7,E2 -21364.7} C_VEL
LIN {X 0,Y 232.036,Z 392.612,A -85,B 0,C 180,E1 -21366.472,E2 -21366.472} C_VEL
LIN {X 0,Y 236.453,Z 381.31,A -85,B 0,C 180,E1 -21367.81,E2 -21367.81} C_VEL
LIN {X 0,Y 240.485,Z 368.804,A -85,B 0,C 180,E1 -21368.927,E2 -21368.927} C_VEL
LIN {X 0,Y 243.81,Z 355.126,A -85,B 0,C 180,E1 -21369.82,E2 -21369.82} C_VEL
LIN {X 0,Y 246.192,Z 340.556,A -85,B 0,C 180,E1 -21370.472,E2 -21370.472} C_VEL
LIN {X 0,Y 249.725,Z 313.456,A -85,B 0,C 180,E1 -21371.601,E2 -21371.601} C_VEL
LIN {X 0,Y 250.052,Z 302.299,A -85,B 0,C 180,E1 -21372.631,E2 -21372.631} C_VEL
LIN {X 0,Y 248.852,Z 298.351,A -85,B 0,C 180,E1 -21373.726,E2 -21373.726} C_VEL
LIN {X 0,Y 246.517,Z 292.476,A -85,B 0,C 180,E1 -21375.911,E2 -21375.911} C_VEL
LIN {X 0,Y 244.158,Z 286.986,A -85,B 0,C 180,E1 -21378.667,E2 -21378.667} C_VEL
LIN {X 0,Y 242.141,Z 282.743,A -85,B 0,C 180,E1 -21382.111,E2 -21382.111} C_VEL
LIN {X 0,Y 241.394,Z 280.763,A -85,B 0,C 180,E1 -21384.608,E2 -21384.608} C_VEL
LIN {X 0,Y 241.187,Z 280.168,A -85,B 0,C 180,E1 -21387.677,E2 -21387.677} C_VEL
LIN {X 0,Y 241.749,Z 280.683,A -85,B 0,C 180,E1 -21390.381,E2 -21390.381} C_VEL
LIN {X 0,Y 243.312,Z 282.778,A -85,B 0,C 180,E1 -21393.564,E2 -21393.564} C_VEL
LIN {X 0,Y 244.28,Z 284.406,A -85,B 0,C 180,E1 -21394.969,E2 -21394.969} C_VEL
LIN {X 0,Y 246.389,Z 287.946,A -85,B 0,C 180,E1 -21397.385,E2 -21397.385} C_VEL
LIN {X 0,Y 248.454,Z 291.997,A -85,B 0,C 180,E1 -21399.371,E2 -21399.371} C_VEL
LIN {X 0,Y 250.769,Z 297.2,A -85,B 0,C 180,E1 -21401.305,E2 -21401.305} C_VEL
LIN {X 0,Y 251.056,Z 297.961,A -85,B 0,C 180,E1 -21401.546,E2 -21401.546} C_VEL
LIN {X 0,Y 245.651,Z 334.799,A -85,B 0,C 180,E1 -21403.268,E2 -21403.268} C_VEL
LIN {X 0,Y 243.087,Z 347.7,A -85,B 0,C 180,E1 -21404.2,E2 -21404.2} C_VEL
LIN {X 0,Y 239.588,Z 360.394,A -85,B 0,C 180,E1 -21405.471,E2 -21405.471} C_VEL
LIN {X 0,Y 235.859,Z 370.921,A -85,B 0,C 180,E1 -21406.867,E2 -21406.867} C_VEL
LIN {X 0,Y 231.557,Z 381.195,A -85,B 0,C 180,E1 -21408.621,E2 -21408.621} C_VEL
LIN {X 0,Y 227.241,Z 389.867,A -85,B 0,C 180,E1 -21410.537,E2 -21410.537} C_VEL
LIN {X 0,Y 222.699,Z 397.593,A -85,B 0,C 180,E1 -21412.747,E2 -21412.747} C_VEL
LIN {X 0,Y 218.106,Z 404.353,A -85,B 0,C 180,E1 -21415.286,E2 -21415.286} C_VEL
LIN {X 0,Y 213.665,Z 409.831,A -85,B 0,C 180,E1 -21418.114,E2 -21418.114} C_VEL
LIN {X 0,Y 210.844,Z 412.754,A -85,B 0,C 180,E1 -21420.171,E2 -21420.171} C_VEL
LIN {X 0,Y 208.699,Z 414.647,A -85,B 0,C 180,E1 -21421.929,E2 -21421.929} C_VEL
LIN {X 0,Y 206.584,Z 416.19,A -85,B 0,C 180,E1 -21423.9,E2 -21423.9} C_VEL
LIN {X 0,Y 204.689,Z 417.202,A -85,B 0,C 180,E1 -21425.911,E2 -21425.911} C_VEL
LIN {X 0,Y 203.069,Z 417.65,A -85,B 0,C 180,E1 -21427.956,E2 -21427.956} C_VEL
LIN {X 0,Y 200.81,Z 417.232,A -85,B 0,C 180,E1 -21431.489,E2 -21431.489} C_VEL
LIN {X 0,Y 199.522,Z 415.834,A -85,B 0,C 180,E1 -21434.274,E2 -21434.274} C_VEL
LIN {X 0,Y 198.613,Z 413.376,A -85,B 0,C 180,E1 -21437.173,E2 -21437.173} C_VEL
LIN {X 0,Y 198.137,Z 408.845,A -85,B 0,C 180,E1 -21440.774,E2 -21440.774} C_VEL
LIN {X 0,Y 198.202,Z 403.093,A -85,B 0,C 180,E1 -21444.064,E2 -21444.064} C_VEL
LIN {X 0,Y 198.621,Z 396.924,A -85,B 0,C 180,E1 -21446.816,E2 -21446.816} C_VEL
LIN {X 0,Y 199.19,Z 389.011,A -85,B 0,C 180,E1 -21449.6,E2 -21449.6} C_VEL
LIN {X 0,Y 199.992,Z 379.775,A -85,B 0,C 180,E1 -21452.194,E2 -21452.194} C_VEL
LIN {X 0,Y 201.002,Z 368.811,A -85,B 0,C 180,E1 -21454.622,E2 -21454.622} C_VEL
LIN {X 0,Y 202.004,Z 357.774,A -85,B 0,C 180,E1 -21456.53,E2 -21456.53} C_VEL
LIN {X 0,Y 202.907,Z 346.276,A -85,B 0,C 180,E1 -21458.073,E2 -21458.073} C_VEL
LIN {X 0,Y 203.675,Z 333.468,A -85,B 0,C 180,E1 -21459.348,E2 -21459.348} C_VEL
LIN {X 0,Y 204.22,Z 320.445,A -85,B 0,C 180,E1 -21460.224,E2 -21460.224} C_VEL
LIN {X 0,Y 206.467,Z 264.162,A -85,B 0,C 180,E1 -21463.127,E2 -21463.127} C_VEL
LIN {X 0,Y 203.23,Z 237.221,A -85,B 0,C 180,E1 -21464.763,E2 -21464.763} C_VEL
LIN {X 0,Y 202.959,Z 235.83,A -85,B 0,C 180,E1 -21465.125,E2 -21465.125} C_VEL
LIN {X 0,Y 201.009,Z 226.067,A -85,B 0,C 180,E1 -21469.037,E2 -21469.037} C_VEL
LIN {X 0,Y 199.758,Z 219.855,A -85,B 0,C 180,E1 -21471.676,E2 -21471.676} C_VEL
LIN {X 0,Y 199.647,Z 219.617,A -85,B 0,C 180,E1 -21474.06,E2 -21474.06} C_VEL
LIN {X 0,Y 199.702,Z 219.609,A -85,B 0,C 180,E1 -21478.136,E2 -21478.136} C_VEL
LIN {X 0,Y 199.686,Z 219.61,A -85,B 0,C 180,E1 -21482.77,E2 -21482.77} C_VEL
LIN {X 0,Y 199.737,Z 219.606,A -85,B 0,C 180,E1 -21487.228,E2 -21487.228} C_VEL
LIN {X 0,Y 199.796,Z 219.596,A -85,B 0,C 180,E1 -21491.756,E2 -21491.756} C_VEL
LIN {X 0,Y 199.847,Z 219.591,A -85,B 0,C 180,E1 -21495.748,E2 -21495.748} C_VEL
LIN {X 0,Y 200.074,Z 219.559,A -85,B 0,C 180,E1 -21499.883,E2 -21499.883} C_VEL
LIN {X 0,Y 200.036,Z 219.566,A -85,B 0,C 180,E1 -21503.948,E2 -21503.948} C_VEL
LIN {X 0,Y 200.32,Z 219.529,A -85,B 0,C 180,E1 -21507.988,E2 -21507.988} C_VEL
LIN {X 0,Y 200.477,Z 219.507,A -85,B 0,C 180,E1 -21509.999,E2 -21509.999} C_VEL
LIN {X 0,Y 200.029,Z 219.567,A -85,B 0,C 180,E1 -21514.028,E2 -21514.028} C_VEL
LIN {X 0,Y 200.108,Z 219.553,A -85,B 0,C 180,E1 -21518.074,E2 -21518.074} C_VEL
LIN {X 0,Y 199.91,Z 219.582,A -85,B 0,C 180,E1 -21522.176,E2 -21522.176} C_VEL
LIN {X 0,Y 199.801,Z 219.593,A -85,B 0,C 180,E1 -21526.342,E2 -21526.342} C_VEL
LIN {X 0,Y 199.696,Z 219.611,A -85,B 0,C 180,E1 -21530.604,E2 -21530.604} C_VEL
LIN {X 0,Y 199.668,Z 219.611,A -85,B 0,C 180,E1 -21534.983,E2 -21534.983} C_VEL
LIN {X 0,Y 199.67,Z 219.612,A -85,B 0,C 180,E1 -21539.521,E2 -21539.521} C_VEL
LIN {X 0,Y 199.659,Z 219.613,A -85,B 0,C 180,E1 -21542.351,E2 -21542.351} C_VEL
LIN {X 0,Y 199.647,Z 219.617,A -85,B 0,C 180,E1 -21546.756,E2 -21546.756} C_VEL
LIN {X 0,Y 199.672,Z 219.61,A -85,B 0,C 180,E1 -21549.311,E2 -21549.311} C_VEL
LIN {X 0,Y 199.656,Z 219.612,A -85,B 0,C 180,E1 -21552.337,E2 -21552.337} C_VEL
LIN {X 0,Y 199.659,Z 219.613,A -85,B 0,C 180,E1 -21555.253,E2 -21555.253} C_VEL
LIN {X 0,Y 199.643,Z 219.616,A -85,B 0,C 180,E1 -21558.023,E2 -21558.023} C_VEL
LIN {X 0,Y 199.67,Z 219.61,A -85,B 0,C 180,E1 -21560.744,E2 -21560.744} C_VEL
LIN {X 0,Y 199.628,Z 219.618,A -85,B 0,C 180,E1 -21565.718,E2 -21565.718} C_VEL
LIN {X 0,Y 199.697,Z 219.607,A -85,B 0,C 180,E1 -21568.138,E2 -21568.138} C_VEL
LIN {X 0,Y 199.68,Z 219.611,A -85,B 0,C 180,E1 -21572.772,E2 -21572.772} C_VEL
LIN {X 0,Y 199.731,Z 219.6,A -85,B 0,C 180,E1 -21577.229,E2 -21577.229} C_VEL
LIN {X 0,Y 199.79,Z 219.599,A -85,B 0,C 180,E1 -21581.758,E2 -21581.758} C_VEL
LIN {X 0,Y 199.829,Z 219.59,A -85,B 0,C 180,E1 -21585.749,E2 -21585.749} C_VEL
LIN {X 0,Y 200.016,Z 219.571,A -85,B 0,C 180,E1 -21589.882,E2 -21589.882} C_VEL
LIN {X 0,Y 200.016,Z 219.568,A -85,B 0,C 180,E1 -21593.95,E2 -21593.95} C_VEL
LIN {X 0,Y 200.315,Z 219.533,A -85,B 0,C 180,E1 -21597.99,E2 -21597.99} C_VEL
LIN {X 0,Y 200.473,Z 219.511,A -85,B 0,C 180,E1 -21600.001,E2 -21600.001} C_VEL
LIN {X 0,Y 200.025,Z 219.568,A -85,B 0,C 180,E1 -21604.031,E2 -21604.031} C_VEL
LIN {X 0,Y 200.114,Z 219.556,A -85,B 0,C 180,E1 -21608.077,E2 -21608.077} C_VEL
LIN {X 0,Y 199.882,Z 219.584,A -85,B 0,C 180,E1 -21612.18,E2 -21612.18} C_VEL
LIN {X 0,Y 199.8,Z 219.595,A -85,B 0,C 180,E1 -21616.345,E2 -21616.345} C_VEL
LIN {X 0,Y 199.696,Z 219.607,A -85,B 0,C 180,E1 -21620.607,E2 -21620.607} C_VEL
LIN {X 0,Y 199.669,Z 219.613,A -85,B 0,C 180,E1 -21624.986,E2 -21624.986} C_VEL
LIN {X 0,Y 199.661,Z 219.615,A -85,B 0,C 180,E1 -21629.526,E2 -21629.526} C_VEL
LIN {X 0,Y 199.668,Z 219.611,A -85,B 0,C 180,E1 -21632.357,E2 -21632.357} C_VEL
LIN {X 0,Y 199.62,Z 219.619,A -85,B 0,C 180,E1 -21636.765,E2 -21636.765} C_VEL
LIN {X 0,Y 199.605,Z 219.622,A -85,B 0,C 180,E1 -21639.33,E2 -21639.33} C_VEL
LIN {X 0,Y 199.57,Z 219.625,A -85,B 0,C 180,E1 -21642.311,E2 -21642.311} C_VEL
LIN {X 0,Y 199.575,Z 219.626,A -85,B 0,C 180,E1 -21645.23,E2 -21645.23} C_VEL
LIN {X 0,Y 199.67,Z 219.789,A -85,B 0,C 180,E1 -21649.519,E2 -21649.519} C_VEL
LIN {X 0,Y 202.426,Z 231.896,A -85,B 0,C 180,E1 -21654.085,E2 -21654.085} C_VEL
LIN {X 0,Y 205.531,Z 246.29,A -85,B 0,C 180,E1 -21659.144,E2 -21659.144} C_VEL
LIN {X 0,Y 205.719,Z 248.084,A -85,B 0,C 180,E1 -21659.743,E2 -21659.743} C_VEL
LIN {X 0,Y 204.414,Z 254.941,A -85,B 0,C 180,E1 -21661.831,E2 -21661.831} C_VEL
LIN {X 0,Y 205.102,Z 277.291,A -85,B 0,C 180,E1 -21662.99,E2 -21662.99} C_VEL
LIN {X 0,Y 205.438,Z 282.429,A -85,B 0,C 180,E1 -21663.258,E2 -21663.258} C_VEL
LIN {X 0,Y 205.03,Z 288.271,A -85,B 0,C 180,E1 -21663.524,E2 -21663.524} C_VEL
LIN {X 0,Y 199.741,Z 309.366,A -85,B 0,C 180,E1 -21664.34,E2 -21664.34} C_VEL
LIN {X 0,Y 199.345,Z 313.281,A -85,B 0,C 180,E1 -21664.52,E2 -21664.52} C_VEL
LIN {X 0,Y 197.764,Z 356.82,A -85,B 0,C 180,E1 -21666.714,E2 -21666.714} C_VEL
LIN {X 0,Y 197.044,Z 368.553,A -85,B 0,C 180,E1 -21667.663,E2 -21667.663} C_VEL
LIN {X 0,Y 196.028,Z 380.311,A -85,B 0,C 180,E1 -21668.992,E2 -21668.992} C_VEL
LIN {X 0,Y 194.836,Z 392.242,A -85,B 0,C 180,E1 -21670.792,E2 -21670.792} C_VEL
LIN {X 0,Y 193.716,Z 402.876,A -85,B 0,C 180,E1 -21672.858,E2 -21672.858} C_VEL
LIN {X 0,Y 192.658,Z 412.494,A -85,B 0,C 180,E1 -21675.207,E2 -21675.207} C_VEL
LIN {X 0,Y 192.059,Z 421.276,A -85,B 0,C 180,E1 -21677.855,E2 -21677.855} C_VEL
LIN {X 0,Y 191.664,Z 429.594,A -85,B 0,C 180,E1 -21681.036,E2 -21681.036} C_VEL
LIN {X 0,Y 191.694,Z 435.142,A -85,B 0,C 180,E1 -21683.687,E2 -21683.687} C_VEL
LIN {X 0,Y 191.956,Z 440.361,A -85,B 0,C 180,E1 -21686.853,E2 -21686.853} C_VEL
LIN {X 0,Y 192.028,Z 444.131,A -85,B 0,C 180,E1 -21690.001,E2 -21690.001} C_VEL
LIN {X 0,Y 191.737,Z 445.88,A -85,B 0,C 180,E1 -21692.102,E2 -21692.102} C_VEL
LIN {X 0,Y 191.296,Z 447.141,A -85,B 0,C 180,E1 -21694.215,E2 -21694.215} C_VEL
LIN {X 0,Y 190.945,Z 447.999,A -85,B 0,C 180,E1 -21696.389,E2 -21696.389} C_VEL
LIN {X 0,Y 190.93,Z 448.397,A -85,B 0,C 180,E1 -21700.607,E2 -21700.607} C_VEL
LIN {X 0,Y 192.065,Z 447.299,A -85,B 0,C 180,E1 -21704.843,E2 -21704.843} C_VEL
LIN {X 0,Y 193.215,Z 446.16,A -85,B 0,C 180,E1 -21706.919,E2 -21706.919} C_VEL
LIN {X 0,Y 196.238,Z 442.69,A -85,B 0,C 180,E1 -21710.987,E2 -21710.987} C_VEL
LIN {X 0,Y 199.209,Z 438.994,A -85,B 0,C 180,E1 -21713.937,E2 -21713.937} C_VEL
LIN {X 0,Y 202.873,Z 434.252,A -85,B 0,C 180,E1 -21716.767,E2 -21716.767} C_VEL
LIN {X 0,Y 208.104,Z 427.204,A -85,B 0,C 180,E1 -21719.878,E2 -21719.878} C_VEL
LIN {X 0,Y 213.15,Z 419.701,A -85,B 0,C 180,E1 -21722.399,E2 -21722.399} C_VEL
LIN {X 0,Y 217.72,Z 412.134,A -85,B 0,C 180,E1 -21724.396,E2 -21724.396} C_VEL
LIN {X 0,Y 222.735,Z 402.991,A -85,B 0,C 180,E1 -21726.273,E2 -21726.273} C_VEL
LIN {X 0,Y 228.196,Z 391.803,A -85,B 0,C 180,E1 -21728.023,E2 -21728.023} C_VEL
LIN {X 0,Y 232.796,Z 380.654,A -85,B 0,C 180,E1 -21729.345,E2 -21729.345} C_VEL
LIN {X 0,Y 237.009,Z 368.214,A -85,B 0,C 180,E1 -21730.441,E2 -21730.441} C_VEL
LIN {X 0,Y 240.48,Z 354.495,A -85,B 0,C 180,E1 -21731.324,E2 -21731.324} C_VEL
LIN {X 0,Y 243.051,Z 339.251,A -85,B 0,C 180,E1 -21732.005,E2 -21732.005} C_VEL
LIN {X 0,Y 246.486,Z 314.826,A -85,B 0,C 180,E1 -21733.036,E2 -21733.036} C_VEL
LIN {X 0,Y 246.884,Z 306.145,A -85,B 0,C 180,E1 -21733.862,E2 -21733.862} C_VEL
LIN {X 0,Y 245.321,Z 301.517,A -85,B 0,C 180,E1 -21735.382,E2 -21735.382} C_VEL
LIN {X 0,Y 243.875,Z 297.756,A -85,B 0,C 180,E1 -21736.973,E2 -21736.973} C_VEL
LIN {X 0,Y 242.318,Z 293.617,A -85,B 0,C 180,E1 -21739.069,E2 -21739.069} C_VEL
LIN {X 0,Y 240.477,Z 289.375,A -85,B 0,C 180,E1 -21742.541,E2 -21742.541} C_VEL
LIN {X 0,Y 239.83,Z 287.517,A -85,B 0,C 180,E1 -21745.137,E2 -21745.137} C_VEL
LIN {X 0,Y 239.777,Z 287.107,A -85,B 0,C 180,E1 -21748.214,E2 -21748.214} C_VEL
LIN {X 0,Y 240.404,Z 287.797,A -85,B 0,C 180,E1 -21750.784,E2 -21750.784} C_VEL
LIN {X 0,Y 242.064,Z 290.276,A -85,B 0,C 180,E1 -21754.026,E2 -21754.026} C_VEL
LIN {X 0,Y 244.242,Z 294.328,A -85,B 0,C 180,E1 -21756.873,E2 -21756.873} C_VEL
LIN {X 0,Y 246.121,Z 298.408,A -85,B 0,C 180,E1 -21758.869,E2 -21758.869} C_VEL
LIN {X 0,Y 247.622,Z 301.854,A -85,B 0,C 180,E1 -21760.211,E2 -21760.211} C_VEL
LIN {X 0,Y 242.294,Z 336.022,A -85,B 0,C 180,E1 -21761.831,E2 -21761.831} C_VEL
LIN {X 0,Y 239.647,Z 348.346,A -85,B 0,C 180,E1 -21762.726,E2 -21762.726} C_VEL
LIN {X 0,Y 235.924,Z 361.213,A -85,B 0,C 180,E1 -21764.004,E2 -21764.004} C_VEL
LIN {X 0,Y 231.694,Z 372.592,A -85,B 0,C 180,E1 -21765.527,E2 -21765.527} C_VEL
LIN {X 0,Y 227.681,Z 381.523,A -85,B 0,C 180,E1 -21767.067,E2 -21767.067} C_VEL
LIN {X 0,Y 222.811,Z 390.641,A -85,B 0,C 180,E1 -21769.09,E2 -21769.09} C_VEL
LIN {X 0,Y 218.185,Z 398.096,A -85,B 0,C 180,E1 -21771.198,E2 -21771.198} C_VEL
LIN {X 0,Y 213.856,Z 404.074,A -85,B 0,C 180,E1 -21773.394,E2 -21773.394} C_VEL
LIN {X 0,Y 209.192,Z 409.638,A -85,B 0,C 180,E1 -21776.146,E2 -21776.146} C_VEL
LIN {X 0,Y 205.024,Z 413.718,A -85,B 0,C 180,E1 -21778.981,E2 -21778.981} C_VEL
LIN {X 0,Y 201.331,Z 416.555,A -85,B 0,C 180,E1 -21782,E2 -21782} C_VEL
LIN {X 0,Y 197.728,Z 418.236,A -85,B 0,C 180,E1 -21785.592,E2 -21785.592} C_VEL
LIN {X 0,Y 195.669,Z 418.461,A -85,B 0,C 180,E1 -21788.259,E2 -21788.259} C_VEL
LIN {X 0,Y 193.642,Z 417.633,A -85,B 0,C 180,E1 -21791.493,E2 -21791.493} C_VEL
LIN {X 0,Y 192.18,Z 415.58,A -85,B 0,C 180,E1 -21794.831,E2 -21794.831} C_VEL
LIN {X 0,Y 191.29,Z 412.161,A -85,B 0,C 180,E1 -21798.241,E2 -21798.241} C_VEL
LIN {X 0,Y 191.007,Z 407.434,A -85,B 0,C 180,E1 -21801.588,E2 -21801.588} C_VEL
LIN {X 0,Y 191.155,Z 402.183,A -85,B 0,C 180,E1 -21804.431,E2 -21804.431} C_VEL
LIN {X 0,Y 191.613,Z 395.561,A -85,B 0,C 180,E1 -21807.288,E2 -21807.288} C_VEL
LIN {X 0,Y 192.233,Z 387.19,A -85,B 0,C 180,E1 -21810.177,E2 -21810.177} C_VEL
LIN {X 0,Y 193.082,Z 377.728,A -85,B 0,C 180,E1 -21812.78,E2 -21812.78} C_VEL
LIN {X 0,Y 193.958,Z 368.572,A -85,B 0,C 180,E1 -21814.797,E2 -21814.797} C_VEL
LIN {X 0,Y 194.99,Z 357.099,A -85,B 0,C 180,E1 -21816.812,E2 -21816.812} C_VEL
LIN {X 0,Y 195.991,Z 344.401,A -85,B 0,C 180,E1 -21818.504,E2 -21818.504} C_VEL
LIN {X 0,Y 196.802,Z 330.381,A -85,B 0,C 180,E1 -21819.832,E2 -21819.832} C_VEL
LIN {X 0,Y 197.508,Z 309.37,A -85,B 0,C 180,E1 -21821.075,E2 -21821.075} C_VEL
LIN {X 0,Y 199.432,Z 264.469,A -85,B 0,C 180,E1 -21823.477,E2 -21823.477} C_VEL
LIN {X 0,Y 196.339,Z 238.571,A -85,B 0,C 180,E1 -21825.096,E2 -21825.096} C_VEL
LIN {X 0,Y 195.911,Z 236.68,A -85,B 0,C 180,E1 -21825.376,E2 -21825.376} C_VEL
LIN {X 0,Y 193.716,Z 225.716,A -85,B 0,C 180,E1 -21829.898,E2 -21829.898} C_VEL
LIN {X 0,Y 192.666,Z 220.674,A -85,B 0,C 180,E1 -21832.156,E2 -21832.156} C_VEL
LIN {X 0,Y 192.611,Z 220.493,A -85,B 0,C 180,E1 -21837.056,E2 -21837.056} C_VEL
LIN {X 0,Y 192.664,Z 220.486,A -85,B 0,C 180,E1 -21841.691,E2 -21841.691} C_VEL
LIN {X 0,Y 192.705,Z 220.479,A -85,B 0,C 180,E1 -21846.347,E2 -21846.347} C_VEL
LIN {X 0,Y 192.731,Z 220.477,A -85,B 0,C 180,E1 -21851.456,E2 -21851.456} C_VEL
LIN {X 0,Y 192.771,Z 220.472,A -85,B 0,C 180,E1 -21855.213,E2 -21855.213} C_VEL
LIN {X 0,Y 193.019,Z 220.439,A -85,B 0,C 180,E1 -21859.509,E2 -21859.509} C_VEL
LIN {X 0,Y 193,Z 220.443,A -85,B 0,C 180,E1 -21863.727,E2 -21863.727} C_VEL
LIN {X 0,Y 193.262,Z 220.408,A -85,B 0,C 180,E1 -21867.915,E2 -21867.915} C_VEL
LIN {X 0,Y 193.441,Z 220.384,A -85,B 0,C 180,E1 -21869.999,E2 -21869.999} C_VEL
LIN {X 0,Y 192.975,Z 220.446,A -85,B 0,C 180,E1 -21874.176,E2 -21874.176} C_VEL
LIN {X 0,Y 193.058,Z 220.431,A -85,B 0,C 180,E1 -21878.371,E2 -21878.371} C_VEL
LIN {X 0,Y 192.849,Z 220.463,A -85,B 0,C 180,E1 -21882.629,E2 -21882.629} C_VEL
LIN {X 0,Y 192.754,Z 220.472,A -85,B 0,C 180,E1 -21886.957,E2 -21886.957} C_VEL
LIN {X 0,Y 192.632,Z 220.489,A -85,B 0,C 180,E1 -21891.396,E2 -21891.396} C_VEL
LIN {X 0,Y 192.66,Z 220.483,A -85,B 0,C 180,E1 -21894.223,E2 -21894.223} C_VEL
LIN {X 0,Y 192.645,Z 220.489,A -85,B 0,C 180,E1 -21898.891,E2 -21898.891} C_VEL
LIN {X 0,Y 192.595,Z 220.489,A -85,B 0,C 180,E1 -21903.184,E2 -21903.184} C_VEL
LIN {X 0,Y 192.594,Z 220.496,A -85,B 0,C 180,E1 -21908.339,E2 -21908.339} C_VEL
LIN {X 0,Y 192.599,Z 220.491,A -85,B 0,C 180,E1 -21913.131,E2 -21913.131} C_VEL
LIN {X 0,Y 192.59,Z 220.494,A -85,B 0,C 180,E1 -21916.87,E2 -21916.87} C_VEL
LIN {X 0,Y 192.591,Z 220.492,A -85,B 0,C 180,E1 -21921.659,E2 -21921.659} C_VEL
LIN {X 0,Y 192.594,Z 220.491,A -85,B 0,C 180,E1 -21926.815,E2 -21926.815} C_VEL
LIN {X 0,Y 192.658,Z 220.486,A -85,B 0,C 180,E1 -21931.692,E2 -21931.692} C_VEL
LIN {X 0,Y 192.699,Z 220.477,A -85,B 0,C 180,E1 -21936.349,E2 -21936.349} C_VEL
LIN {X 0,Y 192.725,Z 220.478,A -85,B 0,C 180,E1 -21941.458,E2 -21941.458} C_VEL
LIN {X 0,Y 192.757,Z 220.469,A -85,B 0,C 180,E1 -21945.214,E2 -21945.214} C_VEL
LIN {X 0,Y 192.939,Z 220.452,A -85,B 0,C 180,E1 -21949.567,E2 -21949.567} C_VEL
LIN {X 0,Y 192.979,Z 220.444,A -85,B 0,C 180,E1 -21953.729,E2 -21953.729} C_VEL
LIN {X 0,Y 193.256,Z 220.413,A -85,B 0,C 180,E1 -21957.917,E2 -21957.917} C_VEL
LIN {X 0,Y 193.437,Z 220.388,A -85,B 0,C 180,E1 -21960.001,E2 -21960.001} C_VEL
LIN {X 0,Y 192.971,Z 220.446,A -85,B 0,C 180,E1 -21964.178,E2 -21964.178} C_VEL
LIN {X 0,Y 193.063,Z 220.433,A -85,B 0,C 180,E1 -21968.374,E2 -21968.374} C_VEL
LIN {X 0,Y 192.805,Z 220.466,A -85,B 0,C 180,E1 -21972.634,E2 -21972.634} C_VEL
LIN {X 0,Y 192.753,Z 220.474,A -85,B 0,C 180,E1 -21976.96,E2 -21976.96} C_VEL
LIN {X 0,Y 192.633,Z 220.49,A -85,B 0,C 180,E1 -21981.399,E2 -21981.399} C_VEL
LIN {X 0,Y 192.66,Z 220.485,A -85,B 0,C 180,E1 -21984.226,E2 -21984.226} C_VEL
LIN {X 0,Y 192.64,Z 220.487,A -85,B 0,C 180,E1 -21988.89,E2 -21988.89} C_VEL
LIN {X 0,Y 192.593,Z 220.495,A -85,B 0,C 180,E1 -21993.188,E2 -21993.188} C_VEL
LIN {X 0,Y 192.548,Z 220.499,A -85,B 0,C 180,E1 -21998.354,E2 -21998.354} C_VEL
LIN {X 0,Y 192.487,Z 220.509,A -85,B 0,C 180,E1 -22003.097,E2 -22003.097} C_VEL
LIN {X 0,Y 192.61,Z 220.599,A -85,B 0,C 180,E1 -22008.984,E2 -22008.984} C_VEL
LIN {X 0,Y 195.024,Z 231.184,A -85,B 0,C 180,E1 -22013.177,E2 -22013.177} C_VEL
LIN {X 0,Y 198.101,Z 245.359,A -85,B 0,C 180,E1 -22018.371,E2 -22018.371} C_VEL
LIN {X 0,Y 198.583,Z 249.212,A -85,B 0,C 180,E1 -22019.716,E2 -22019.716} C_VEL
LIN {X 0,Y 197.499,Z 254.386,A -85,B 0,C 180,E1 -22021.363,E2 -22021.363} C_VEL
LIN {X 0,Y 197.748,Z 270.585,A -85,B 0,C 180,E1 -22022.269,E2 -22022.269} C_VEL
LIN {X 0,Y 199.758,Z 303.56,A -85,B 0,C 180,E1 -22024.052,E2 -22024.052} C_VEL
LIN {X 0,Y 199.345,Z 313.281,A -85,B 0,C 180,E1 -22024.52,E2 -22024.52} C_VEL
LIN {X 0,Y 198.453,Z 319.058,A -85,B 0,C 180,E1 -22024.774,E2 -22024.774} C_VEL
LIN {X 0,Y 192.006,Z 337.672,A -85,B 0,C 180,E1 -22025.484,E2 -22025.484} C_VEL
LIN {X 0,Y 191.174,Z 343.448,A -85,B 0,C 180,E1 -22025.757,E2 -22025.757} C_VEL
LIN {X 0,Y 190.656,Z 358.738,A -85,B 0,C 180,E1 -22026.657,E2 -22026.657} C_VEL
LIN {X 0,Y 189.811,Z 370.224,A -85,B 0,C 180,E1 -22027.699,E2 -22027.699} C_VEL
LIN {X 0,Y 188.78,Z 381.852,A -85,B 0,C 180,E1 -22029.143,E2 -22029.143} C_VEL
LIN {X 0,Y 187.686,Z 392.561,A -85,B 0,C 180,E1 -22030.876,E2 -22030.876} C_VEL
LIN {X 0,Y 186.423,Z 404.103,A -85,B 0,C 180,E1 -22033.296,E2 -22033.296} C_VEL
LIN {X 0,Y 185.509,Z 413.401,A -85,B 0,C 180,E1 -22035.746,E2 -22035.746} C_VEL
LIN {X 0,Y 184.91,Z 421.775,A -85,B 0,C 180,E1 -22038.492,E2 -22038.492} C_VEL
LIN {X 0,Y 184.664,Z 429.651,A -85,B 0,C 180,E1 -22041.703,E2 -22041.703} C_VEL
LIN {X 0,Y 184.767,Z 435.202,A -85,B 0,C 180,E1 -22044.545,E2 -22044.545} C_VEL
LIN {X 0,Y 185.012,Z 440.177,A -85,B 0,C 180,E1 -22047.825,E2 -22047.825} C_VEL
LIN {X 0,Y 185.069,Z 442.692,A -85,B 0,C 180,E1 -22050.002,E2 -22050.002} C_VEL
LIN {X 0,Y 184.731,Z 444.616,A -85,B 0,C 180,E1 -22052.182,E2 -22052.182} C_VEL
LIN {X 0,Y 184.275,Z 445.993,A -85,B 0,C 180,E1 -22054.376,E2 -22054.376} C_VEL
LIN {X 0,Y 183.786,Z 447.451,A -85,B 0,C 180,E1 -22058.8,E2 -22058.8} C_VEL
LIN {X 0,Y 183.924,Z 447.612,A -85,B 0,C 180,E1 -22061.016,E2 -22061.016} C_VEL
LIN {X 0,Y 185.188,Z 446.737,A -85,B 0,C 180,E1 -22065.407,E2 -22065.407} C_VEL
LIN {X 0,Y 187.837,Z 444.39,A -85,B 0,C 180,E1 -22069.68,E2 -22069.68} C_VEL
LIN {X 0,Y 191.643,Z 440.392,A -85,B 0,C 180,E1 -22073.792,E2 -22073.792} C_VEL
LIN {X 0,Y 195.213,Z 436.276,A -85,B 0,C 180,E1 -22076.746,E2 -22076.746} C_VEL
LIN {X 0,Y 200.395,Z 430.146,A -85,B 0,C 180,E1 -22079.985,E2 -22079.985} C_VEL
LIN {X 0,Y 205.468,Z 423.471,A -85,B 0,C 180,E1 -22082.598,E2 -22082.598} C_VEL
LIN {X 0,Y 211.047,Z 415.292,A -85,B 0,C 180,E1 -22085.061,E2 -22085.061} C_VEL
LIN {X 0,Y 216.119,Z 407.107,A -85,B 0,C 180,E1 -22086.986,E2 -22086.986} C_VEL
LIN {X 0,Y 221.606,Z 397.102,A -85,B 0,C 180,E1 -22088.783,E2 -22088.783} C_VEL
LIN {X 0,Y 226.918,Z 385.956,A -85,B 0,C 180,E1 -22090.282,E2 -22090.282} C_VEL
LIN {X 0,Y 231.788,Z 373.461,A -85,B 0,C 180,E1 -22091.551,E2 -22091.551} C_VEL
LIN {X 0,Y 235.602,Z 361.414,A -85,B 0,C 180,E1 -22092.448,E2 -22092.448} C_VEL
LIN {X 0,Y 238.774,Z 347.733,A -85,B 0,C 180,E1 -22093.182,E2 -22093.182} C_VEL
LIN {X 0,Y 243.489,Z 316.3,A -85,B 0,C 180,E1 -22094.508,E2 -22094.508} C_VEL
LIN {X 0,Y 243.838,Z 310.396,A -85,B 0,C 180,E1 -22095.075,E2 -22095.075} C_VEL
LIN {X 0,Y 242.222,Z 305.161,A -85,B 0,C 180,E1 -22097.006,E2 -22097.006} C_VEL
LIN {X 0,Y 240.36,Z 300.034,A -85,B 0,C 180,E1 -22099.65,E2 -22099.65} C_VEL
LIN {X 0,Y 238.797,Z 296.021,A -85,B 0,C 180,E1 -22102.991,E2 -22102.991} C_VEL
LIN {X 0,Y 238.312,Z 294.423,A -85,B 0,C 180,E1 -22105.278,E2 -22105.278} C_VEL
LIN {X 0,Y 238.233,Z 294.034,A -85,B 0,C 180,E1 -22107.925,E2 -22107.925} C_VEL
LIN {X 0,Y 238.794,Z 294.665,A -85,B 0,C 180,E1 -22110.568,E2 -22110.568} C_VEL
LIN {X 0,Y 240.201,Z 296.857,A -85,B 0,C 180,E1 -22113.583,E2 -22113.583} C_VEL
LIN {X 0,Y 242.249,Z 301.066,A -85,B 0,C 180,E1 -22116.523,E2 -22116.523} C_VEL
LIN {X 0,Y 244.01,Z 305.045,A -85,B 0,C 180,E1 -22118.484,E2 -22118.484} C_VEL
LIN {X 0,Y 244.322,Z 306.094,A -85,B 0,C 180,E1 -22118.862,E2 -22118.862} C_VEL
LIN {X 0,Y 239.298,Z 336.866,A -85,B 0,C 180,E1 -22120.314,E2 -22120.314} C_VEL
LIN {X 0,Y 236.38,Z 349.739,A -85,B 0,C 180,E1 -22121.247,E2 -22121.247} C_VEL
LIN {X 0,Y 232.722,Z 361.571,A -85,B 0,C 180,E1 -22122.422,E2 -22122.422} C_VEL
LIN {X 0,Y 228.288,Z 372.827,A -85,B 0,C 180,E1 -22123.914,E2 -22123.914} C_VEL
LIN {X 0,Y 223.467,Z 382.974,A -85,B 0,C 180,E1 -22125.66,E2 -22125.66} C_VEL
LIN {X 0,Y 218.821,Z 391.205,A -85,B 0,C 180,E1 -22127.478,E2 -22127.478} C_VEL
LIN {X 0,Y 213.813,Z 398.786,A -85,B 0,C 180,E1 -22129.646,E2 -22129.646} C_VEL
LIN {X 0,Y 208.408,Z 405.695,A -85,B 0,C 180,E1 -22132.247,E2 -22132.247} C_VEL
LIN {X 0,Y 203.466,Z 411.059,A -85,B 0,C 180,E1 -22135.044,E2 -22135.044} C_VEL
LIN {X 0,Y 198.99,Z 414.986,A -85,B 0,C 180,E1 -22137.975,E2 -22137.975} C_VEL
LIN {X 0,Y 196.338,Z 416.866,A -85,B 0,C 180,E1 -22139.999,E2 -22139.999} C_VEL
LIN {X 0,Y 193.915,Z 418.218,A -85,B 0,C 180,E1 -22142.076,E2 -22142.076} C_VEL
LIN {X 0,Y 190.617,Z 419.249,A -85,B 0,C 180,E1 -22145.437,E2 -22145.437} C_VEL
LIN {X 0,Y 188.245,Z 419.041,A -85,B 0,C 180,E1 -22148.587,E2 -22148.587} C_VEL
LIN {X 0,Y 186.491,Z 417.924,A -85,B 0,C 180,E1 -22151.525,E2 -22151.525} C_VEL
LIN {X 0,Y 184.885,Z 415.077,A -85,B 0,C 180,E1 -22155.431,E2 -22155.431} C_VEL
LIN {X 0,Y 184.098,Z 411.121,A -85,B 0,C 180,E1 -22158.934,E2 -22158.934} C_VEL
LIN {X 0,Y 183.914,Z 405.729,A -85,B 0,C 180,E1 -22162.465,E2 -22162.465} C_VEL
LIN {X 0,Y 184.184,Z 399.842,A -85,B 0,C 180,E1 -22165.42,E2 -22165.42} C_VEL
LIN {X 0,Y 184.692,Z 392.718,A -85,B 0,C 180,E1 -22168.294,E2 -22168.294} C_VEL
LIN {X 0,Y 185.402,Z 384.096,A -85,B 0,C 180,E1 -22171.095,E2 -22171.095} C_VEL
LIN {X 0,Y 186.383,Z 373.691,A -85,B 0,C 180,E1 -22173.787,E2 -22173.787} C_VEL
LIN {X 0,Y 187.477,Z 361.791,A -85,B 0,C 180,E1 -22176.186,E2 -22176.186} C_VEL
LIN {X 0,Y 188.609,Z 348.93,A -85,B 0,C 180,E1 -22178.153,E2 -22178.153} C_VEL
LIN {X 0,Y 189.472,Z 335.947,A -85,B 0,C 180,E1 -22179.606,E2 -22179.606} C_VEL
LIN {X 0,Y 190.075,Z 322.498,A -85,B 0,C 180,E1 -22180.623,E2 -22180.623} C_VEL
LIN {X 0,Y 192.472,Z 265.192,A -85,B 0,C 180,E1 -22183.819,E2 -22183.819} C_VEL
LIN {X 0,Y 189.638,Z 240.576,A -85,B 0,C 180,E1 -22185.415,E2 -22185.415} C_VEL
LIN {X 0,Y 188.814,Z 237.247,A -85,B 0,C 180,E1 -22185.739,E2 -22185.739} C_VEL
LIN {X 0,Y 186.393,Z 225.131,A -85,B 0,C 180,E1 -22190.903,E2 -22190.903} C_VEL
LIN {X 0,Y 185.592,Z 221.482,A -85,B 0,C 180,E1 -22192.675,E2 -22192.675} C_VEL
LIN {X 0,Y 185.546,Z 221.373,A -85,B 0,C 180,E1 -22197.974,E2 -22197.974} C_VEL
